	                  IF #coordSystem = #INDEX_COORDSYSTEM_TCS THEN
	                    #instMC_MoveLinearRelative.CoordSystem := "CS_WCS";
	                    IF #jogDirection < #JOG_DIRECTION_A THEN
	                      "LKinCtrl_OcsToWcs"(ocsX      := 0,
	                                          ocsY      := 0,
	                                          ocsZ      := 0,
	                                          ocsA      := #axesGroup.TcpInWcs.a.Position,
	                                          ocsB      := #axesGroup.TcpInWcs.b.Position,
	                                          ocsC      := #axesGroup.TcpInWcs.c.Position,
	                                          pointXOcs := #instMC_MoveLinearRelative.Distance[1],
	                                          pointYOcs := #instMC_MoveLinearRelative.Distance[2],
	                                          pointZOcs := #instMC_MoveLinearRelative.Distance[3],
	                                          pointAOcs := #instMC_MoveLinearRelative.Distance[4],
	                                          pointBOcs := #instMC_MoveLinearRelative.Distance[5],
	                                          pointCOcs := #instMC_MoveLinearRelative.Distance[6],
	                                          pointXWcs => #instMC_MoveLinearRelative.Distance[1],
	                                          pointYWcs => #instMC_MoveLinearRelative.Distance[2],
	                                          pointZWcs => #instMC_MoveLinearRelative.Distance[3],
	                                          pointAWcs => #instMC_MoveLinearRelative.Distance[4],
	                                          pointBWcs => #instMC_MoveLinearRelative.Distance[5],
	                                          pointCWcs => #instMC_MoveLinearRelative.Distance[6]);
	                      
	                      // reset rotation due to numeric inaccuracy of frame trans
	                      FOR #tempCounter := 4 TO 6 DO
	                        #instMC_MoveLinearRelative.Distance[#tempCounter] := 0.0;
	                      END_FOR;
	                    END_IF;
	                  ELSIF (#coordSystem >= "LKINCTRL_CS_NO_OF_FIRST_USER_FRAME" AND #coordSystem <= "LKINCTRL_CS_NO_OF_LAST_USER_FRAME") THEN
	                    #instMC_MoveLinearRelative.CoordSystem := "CS_WCS";
	                    IF #jogDirection < #JOG_DIRECTION_A THEN
	                      "LKinCtrl_OcsToWcs"(ocsX      := 0,
	                                          ocsY      := 0,
	                                          ocsZ      := 0,
	                                          ocsA      := #userFrames[#coordSystem].a,
	                                          ocsB      := #userFrames[#coordSystem].b,
	                                          ocsC      := #userFrames[#coordSystem].c,
	                                          pointXOcs := #instMC_MoveLinearRelative.Distance[1],
	                                          pointYOcs := #instMC_MoveLinearRelative.Distance[2],
	                                          pointZOcs := #instMC_MoveLinearRelative.Distance[3],
	                                          pointAOcs := #instMC_MoveLinearRelative.Distance[4],
	                                          pointBOcs := #instMC_MoveLinearRelative.Distance[5],
	                                          pointCOcs := #instMC_MoveLinearRelative.Distance[6],
	                                          pointXWcs => #instMC_MoveLinearRelative.Distance[1],
	                                          pointYWcs => #instMC_MoveLinearRelative.Distance[2],
	                                          pointZWcs => #instMC_MoveLinearRelative.Distance[3],
	                                          pointAWcs => #instMC_MoveLinearRelative.Distance[4],
	                                          pointBWcs => #instMC_MoveLinearRelative.Distance[5],
	                                          pointCWcs => #instMC_MoveLinearRelative.Distance[6]);
	                      
	                      // reset rotation due to numeric inaccuracy of frame trans
	                      FOR #tempCounter := 4 TO 6 DO
	                        #instMC_MoveLinearRelative.Distance[#tempCounter] := 0.0;
	                      END_FOR;
	                    END_IF;
	                  END_IF;
	                END_IF;
	                
	              #JOG_DIRECTION_RZ..#JOG_DIRECTION_RX: // Jogging around A,B,C
	                // set MC_MoveLinearAbsolute parameter
	                #instMC_MoveLinearAbsolute.Velocity := #dynamics.path.velocity;
	                #instMC_MoveLinearAbsolute.Acceleration := #dynamics.path.acceleration;
	                #instMC_MoveLinearAbsolute.Deceleration := #dynamics.path.deceleration;
	                #instMC_MoveLinearAbsolute.Jerk := #dynamics.path.jerk;
	                
	                // read current position and rotation matrix
	                CASE #coordSystem OF
	                  "CS_WCS", #INDEX_COORDSYSTEM_TCS: // in WCS and TCS
	                    // get rotation matrix representation of current position
	                    "LKinCtrl_RotXYZ"(angleA       := #axesGroup.TcpInWcs.a.Position,
	                                      angleB       := #axesGroup.TcpInWcs.b.Position,
	                                      angleC       := #axesGroup.TcpInWcs.c.Position,
	                                      resultMatrix := #statRotMatrix1);
	                    
	                    // do not move translatory
	                    #instMC_MoveLinearAbsolute.CoordSystem := "CS_WCS";
	                    #instMC_MoveLinearAbsolute.Position[1] := #axesGroup.TcpInWcs.x.Position;
	                    #instMC_MoveLinearAbsolute.Position[2] := #axesGroup.TcpInWcs.y.Position;
	                    #instMC_MoveLinearAbsolute.Position[3] := #axesGroup.TcpInWcs.z.Position;
	                  "CS_OCS1".."CS_OCS3": // OCS 1-3
	                    // get rotation matrix representation of current position
	                    "LKinCtrl_RotXYZ"(angleA       := #axesGroup.TcpInOcs[#coordSystem].a.Position,
	                                      angleB       := #axesGroup.TcpInOcs[#coordSystem].b.Position,
	                                      angleC       := #axesGroup.TcpInOcs[#coordSystem].c.Position,
	                                      resultMatrix := #statRotMatrix1);
	                    
	                    // do not move translatory
	                    #instMC_MoveLinearAbsolute.CoordSystem := #coordSystem;
	                    #instMC_MoveLinearAbsolute.Position[1] := #axesGroup.TcpInOcs[#coordSystem].x.Position;
	                    #instMC_MoveLinearAbsolute.Position[2] := #axesGroup.TcpInOcs[#coordSystem].y.Position;
	                    #instMC_MoveLinearAbsolute.Position[3] := #axesGroup.TcpInOcs[#coordSystem].z.Position;
	                  "LKINCTRL_CS_NO_OF_FIRST_USER_FRAME".."LKINCTRL_CS_NO_OF_LAST_USER_FRAME": // UCS
	                    // Calculate current UCS position 
	                    "LKinCtrl_WcsToOcs"(ocsX      := #userFrames[#coordSystem].x,
	                                        ocsY      := #userFrames[#coordSystem].y,
	                                        ocsZ      := #userFrames[#coordSystem].z,
	                                        ocsA      := #userFrames[#coordSystem].a,
	                                        ocsB      := #userFrames[#coordSystem].b,
	                                        ocsC      := #userFrames[#coordSystem].c,
	                                        pointXWcs := #axesGroup.TcpInWcs.x.Position,
	                                        pointYWcs := #axesGroup.TcpInWcs.y.Position,
	                                        pointZWcs := #axesGroup.TcpInWcs.z.Position,
	                                        pointAWcs := #axesGroup.TcpInWcs.a.Position,
	                                        pointBWcs := #axesGroup.TcpInWcs.b.Position,
	                                        pointCWcs := #axesGroup.TcpInWcs.c.Position,
	                                        pointXOcs => #tempTcpInUcs[1],
	                                        pointYOcs => #tempTcpInUcs[2],
	                                        pointZOcs => #tempTcpInUcs[3],
	                                        pointAOcs => #tempTcpInUcs[4],
	                                        pointBOcs => #tempTcpInUcs[5],
	                                        pointCOcs => #tempTcpInUcs[6]);
	                    
	                    // get rotation matrix representation of current position
	                    "LKinCtrl_RotXYZ"(angleA       := #tempTcpInUcs[4],
	                                      angleB       := #tempTcpInUcs[5],
	                                      angleC       := #tempTcpInUcs[6],
	                                      resultMatrix := #statRotMatrix1);
	                    
	                    // do not move translatory
	                    #instMC_MoveLinearAbsolute.CoordSystem := "CS_WCS";
	                    #instMC_MoveLinearAbsolute.Position[1] := #axesGroup.TcpInWcs.x.Position;
	                    #instMC_MoveLinearAbsolute.Position[2] := #axesGroup.TcpInWcs.y.Position;
	                    #instMC_MoveLinearAbsolute.Position[3] := #axesGroup.TcpInWcs.z.Position;
	                END_CASE;
	                
	                // Get rotation matrix based on direction and distance
	                CASE #jogDirection OF
	                  #JOG_DIRECTION_RZ:
	                    "LKinCtrl_RotZ"(angle     := #tempJogDistance,
	                                    rotMatrix := #statRotMatrix2);
	                  #JOG_DIRECTION_RY:
	                    "LKinCtrl_RotY"(angle     := #tempJogDistance,
	                                    rotMatrix := #statRotMatrix2);
	                  #JOG_DIRECTION_RX:
	                    "LKinCtrl_RotX"(angle     := #tempJogDistance,
	                                    rotMatrix := #statRotMatrix2);
	                END_CASE;
	                
	                // Calculate rotation matrix for target orientation
	                IF #coordSystem = #INDEX_COORDSYSTEM_TCS THEN
	                  // Calc rotation matrix TCS
	                  "LKinCtrl_MatrixMultiplication"(error        => #tempError,
	                                                  status       => #tempRetStatus,
	                                                  matrix1      := #statRotMatrix1,
	                                                  matrix2      := #statRotMatrix2,
	                                                  matrixResult := #statRotMatrix3);
	                ELSE
	                  // Calc rotation matrix regular
	                  "LKinCtrl_MatrixMultiplication"(error        => #tempError,
	                                                  status       => #tempRetStatus,
	                                                  matrix1      := #statRotMatrix2,
	                                                  matrix2      := #statRotMatrix1,
	                                                  matrixResult := #statRotMatrix3);
	                END_IF;
	                
	                // Assign target orientation to MC_MoveLinearAbsolute
	                IF #coordSystem >= "LKINCTRL_CS_NO_OF_FIRST_USER_FRAME" AND #coordSystem <= "LKINCTRL_CS_NO_OF_LAST_USER_FRAME" THEN
	                  // calculate rotated target position in UCS
	                  "LKinCtrl_InvRotXYZ"(A         => #tempTcpInUcs[4],
	                                       B         => #tempTcpInUcs[5],
	                                       C         => #tempTcpInUcs[6],
	                                       rotMatrix := #statRotMatrix3);
	                  
	                  // Calculate target WCS position since coordinate system of UCS for system is WCS
	                  "LKinCtrl_OcsToWcs"(ocsX      := #userFrames[#coordSystem].x,
	                                      ocsY      := #userFrames[#coordSystem].y,
	                                      ocsZ      := #userFrames[#coordSystem].z,
	                                      ocsA      := #userFrames[#coordSystem].a,
	                                      ocsB      := #userFrames[#coordSystem].b,
	                                      ocsC      := #userFrames[#coordSystem].c,
	                                      pointXOcs := #tempTcpInUcs[1],
	                                      pointYOcs := #tempTcpInUcs[2],
	                                      pointZOcs := #tempTcpInUcs[3],
	                                      pointAOcs := #tempTcpInUcs[4],
	                                      pointBOcs := #tempTcpInUcs[5],
	                                      pointCOcs := #tempTcpInUcs[6],
	                                      pointXWcs => #tempTcpInUcs[1], // dummy
	                                      pointYWcs => #tempTcpInUcs[2], // dummy
	                                      pointZWcs => #tempTcpInUcs[3], // dummy
	                                      pointAWcs => #instMC_MoveLinearAbsolute.Position[4],
	                                      pointBWcs => #instMC_MoveLinearAbsolute.Position[5],
	                                      pointCWcs => #instMC_MoveLinearAbsolute.Position[6]);
	                  
	                ELSE
	                  // calculate rotated target position
	                  "LKinCtrl_InvRotXYZ"(A         => #instMC_MoveLinearAbsolute.Position[4],
	                                       B         => #instMC_MoveLinearAbsolute.Position[5],
	                                       C         => #instMC_MoveLinearAbsolute.Position[6],
	                                       rotMatrix := #statRotMatrix3);
	                END_IF;
	                
	                // 3D + A,B plausibility check for C
	                IF #statTypeOfKinematics = 26 OR #statTypeOfKinematics = 27 OR #statTypeOfKinematics = 35 THEN
	                  // Check if C is around 0.0 or +-180.0
	                  IF ABS(180.0 - #instMC_MoveLinearAbsolute.Position[6]) < #TOLERANCE_C THEN // Check +180°
	                    #instMC_MoveLinearAbsolute.Position[6] := 180.0;
	                  ELSIF ABS(-180.0 - #instMC_MoveLinearAbsolute.Position[6]) < #TOLERANCE_C THEN // Check -180°
	                    #instMC_MoveLinearAbsolute.Position[6] := -180.0;
	                  ELSIF ABS(#instMC_MoveLinearAbsolute.Position[6]) < #TOLERANCE_C THEN // Check 0.0
	                    #instMC_MoveLinearAbsolute.Position[6] := 0.0;
	                  ELSE
	                    // error wrong value for C
	                    #statStatus := #ERR_JOG_DIRECTION_NOT_POSSIBLE;
	                  END_IF;
	                END_IF;
	                
	            END_CASE;
	            
	          END_REGION
	            // jog to position
	            //*********************************************************************************************************
	        ELSIF #tempJogToPosition THEN
	          REGION JOG_TO_TARGET_LINEAR
	            // set jog target position and configuration
	            #instMC_MoveLinearAbsolute.Position[1] := #targetPosition.x;
	            #instMC_MoveLinearAbsolute.Position[2] := #targetPosition.y;
	            #instMC_MoveLinearAbsolute.Position[3] := #targetPosition.z;
	            #instMC_MoveLinearAbsolute.Position[4] := #targetPosition.a;
	            #instMC_MoveLinearAbsolute.Position[5] := #targetPosition.b;
	            #instMC_MoveLinearAbsolute.Position[6] := #targetPosition.c;
	            #instMC_MoveLinearAbsolute.CoordSystem := #coordSystem;
	            // convert from UCS to WCS if necessary
	            IF (#coordSystem >= "LKINCTRL_CS_NO_OF_FIRST_USER_FRAME" AND #coordSystem <= "LKINCTRL_CS_NO_OF_LAST_USER_FRAME") THEN
	              #instMC_MoveLinearAbsolute.CoordSystem := "CS_WCS";
	              "LKinCtrl_OcsToWcs"(ocsX      := #userFrames[#coordSystem].x,
	                                  ocsY      := #userFrames[#coordSystem].y,
	                                  ocsZ      := #userFrames[#coordSystem].z,
	                                  ocsA      := #userFrames[#coordSystem].a,
	                                  ocsB      := #userFrames[#coordSystem].b,
	                                  ocsC      := #userFrames[#coordSystem].c,
	                                  pointXOcs := #targetPosition.x,
	                                  pointYOcs := #targetPosition.y,
	                                  pointZOcs := #targetPosition.z,
	                                  pointAOcs := #targetPosition.a,
	                                  pointBOcs := #targetPosition.b,
	                                  pointCOcs := #targetPosition.c,
	                                  pointXWcs => #instMC_MoveLinearAbsolute.Position[1],
	                                  pointYWcs => #instMC_MoveLinearAbsolute.Position[2],
	                                  pointZWcs => #instMC_MoveLinearAbsolute.Position[3],
	                                  pointAWcs => #instMC_MoveLinearAbsolute.Position[4],
	                                  pointBWcs => #instMC_MoveLinearAbsolute.Position[5],
	                                  pointCWcs => #instMC_MoveLinearAbsolute.Position[6]);
	            END_IF;
	            // convert from TCS to WCS if necessary
	            IF #coordSystem = #INDEX_COORDSYSTEM_TCS THEN
	              #instMC_MoveLinearAbsolute.CoordSystem := "CS_WCS";
	              "LKinCtrl_OcsToWcs"(ocsX      := #axesGroup.TcpInWcs.x.Position,
	                                  ocsY      := #axesGroup.TcpInWcs.y.Position,
	                                  ocsZ      := #axesGroup.TcpInWcs.z.Position,
	                                  ocsA      := #axesGroup.TcpInWcs.a.Position,
	                                  ocsB      := #axesGroup.TcpInWcs.b.Position,
	                                  ocsC      := #axesGroup.TcpInWcs.c.Position,
	                                  pointXOcs := #instMC_MoveLinearAbsolute.Position[1],
	                                  pointYOcs := #instMC_MoveLinearAbsolute.Position[2],
	                                  pointZOcs := #instMC_MoveLinearAbsolute.Position[3],
	                                  pointAOcs := #instMC_MoveLinearAbsolute.Position[4],
	                                  pointBOcs := #instMC_MoveLinearAbsolute.Position[5],
	                                  pointCOcs := #instMC_MoveLinearAbsolute.Position[6],
	                                  pointXWcs => #instMC_MoveLinearAbsolute.Position[1],
	                                  pointYWcs => #instMC_MoveLinearAbsolute.Position[2],
	                                  pointZWcs => #instMC_MoveLinearAbsolute.Position[3],
	                                  pointAWcs => #instMC_MoveLinearAbsolute.Position[4],
	                                  pointBWcs => #instMC_MoveLinearAbsolute.Position[5],
	                                  pointCWcs => #instMC_MoveLinearAbsolute.Position[6]);
	            END_IF;
	            
	            #instMC_MoveLinearAbsolute.Velocity := #dynamics.path.velocity;
	            #instMC_MoveLinearAbsolute.Acceleration := #dynamics.path.acceleration;
	            #instMC_MoveLinearAbsolute.Deceleration := #dynamics.path.deceleration;
	            #instMC_MoveLinearAbsolute.Jerk := #dynamics.path.jerk;
	            #instMC_MoveLinearAbsolute.DynamicAdaption := #dynamics.dynamicAdaption;
	            #instMC_MoveLinearAbsolute.DirectionA := #dynamics.directionA;
	          END_REGION
	            // jog synchronous point to point
	            //*********************************************************************************************************
	        ELSIF #tempJogSPTP THEN
	          REGION JOG_TO_POS_SPTP
	            #instMC_MoveDirectAbsolute.Position[1] := #targetPosition.x;
	            #instMC_MoveDirectAbsolute.Position[2] := #targetPosition.y;
	            #instMC_MoveDirectAbsolute.Position[3] := #targetPosition.z;
	            #instMC_MoveDirectAbsolute.Position[4] := #targetPosition.a;
	            #instMC_MoveDirectAbsolute.Position[5] := #targetPosition.b;
	            #instMC_MoveDirectAbsolute.Position[6] := #targetPosition.c;
	            #instMC_MoveDirectAbsolute.CoordSystem := #coordSystem;
	            // convert from UCS to WCS if necessary
	            IF (#coordSystem >= "LKINCTRL_CS_NO_OF_FIRST_USER_FRAME" AND #coordSystem <= "LKINCTRL_CS_NO_OF_LAST_USER_FRAME") THEN
	              #instMC_MoveDirectAbsolute.CoordSystem := "CS_WCS";
	              "LKinCtrl_OcsToWcs"(ocsX      := #userFrames[#coordSystem].x,
	                                  ocsY      := #userFrames[#coordSystem].y,
	                                  ocsZ      := #userFrames[#coordSystem].z,
	                                  ocsA      := #userFrames[#coordSystem].a,
	                                  ocsB      := #userFrames[#coordSystem].b,
	                                  ocsC      := #userFrames[#coordSystem].c,
	                                  pointXOcs := #targetPosition.x,
	                                  pointYOcs := #targetPosition.y,
	                                  pointZOcs := #targetPosition.z,
	                                  pointAOcs := #targetPosition.a,
	                                  pointBOcs := #targetPosition.b,
	                                  pointCOcs := #targetPosition.c,
	                                  pointXWcs => #instMC_MoveDirectAbsolute.Position[1],
	                                  pointYWcs => #instMC_MoveDirectAbsolute.Position[2],
	                                  pointZWcs => #instMC_MoveDirectAbsolute.Position[3],
	                                  pointAWcs => #instMC_MoveDirectAbsolute.Position[4],
	                                  pointBWcs => #instMC_MoveDirectAbsolute.Position[5],
	                                  pointCWcs => #instMC_MoveDirectAbsolute.Position[6]);
	            END_IF;
	            
	            #instMC_MoveDirectAbsolute.VelocityFactor := #dynamics.sPTP.velocityFactor;
	            #instMC_MoveDirectAbsolute.AccelerationFactor := #dynamics.sPTP.accelerationFactor;
	            #instMC_MoveDirectAbsolute.DecelerationFactor := #dynamics.sPTP.decelerationFactor;
	            #instMC_MoveDirectAbsolute.JerkFactor := #dynamics.sPTP.jerkFactor;
	            #instMC_MoveDirectAbsolute.LinkConstellation := #linkconstellation;
	            #instMC_MoveDirectAbsolute.PositionMode := 1;
	            #instMC_MoveDirectAbsolute.DirectionA := #dynamics.directionA;
	            #instMC_MoveDirectAbsolute.TurnJoint := #turnJoint;
	          END_REGION
	          END_IF;
	        END_REGION
	        
	        REGION SET_ORIENTATION_DYNAMICS
	          IF (((#jogDirection >= #JOG_DIRECTION_A AND #jogDirection <= #JOG_DIRECTION_RX) AND (#tempJogForward OR #tempJogBackward)) OR #tempJogToPosition)
	            AND (#dynamics.orientation.velocity > 0.0 // check if change of orientation dynamics is required
	            OR #dynamics.orientation.acceleration > 0.0
	            OR #dynamics.orientation.deceleration > 0.0
	            OR #dynamics.orientation.jerk > 0.0)
	          THEN
	            // safe default dynamics for orientation axis
	            #statOrientationDynamicsOld.velocity := #axesGroup.DynamicDefaults.Orientation.Velocity;
	            #statOrientationDynamicsOld.acceleration := #axesGroup.DynamicDefaults.Orientation.Acceleration;
	            #statOrientationDynamicsOld.deceleration := #axesGroup.DynamicDefaults.Orientation.Deceleration;
	            #statOrientationDynamicsOld.jerk := #axesGroup.DynamicDefaults.Orientation.Jerk;
	            
	            // change orientation default dynamics temporary
	            IF #dynamics.orientation.velocity > 0.0 THEN
	              #axesGroup.DynamicDefaults.Orientation.Velocity := #dynamics.orientation.velocity;
	            END_IF;
	            IF #dynamics.orientation.acceleration > 0.0 THEN
	              #axesGroup.DynamicDefaults.Orientation.Acceleration := #dynamics.orientation.acceleration;
	            END_IF;
	            IF #dynamics.orientation.deceleration > 0.0 THEN
	              #axesGroup.DynamicDefaults.Orientation.Deceleration := #dynamics.orientation.deceleration;
	            END_IF;
	            IF #dynamics.orientation.jerk > 0.0 THEN
	              #axesGroup.DynamicDefaults.Orientation.Jerk := #dynamics.orientation.jerk;
	            END_IF;
	            
	            // Orientation default dynamics will be reseted to previous values after jogging
	            #statOrientationDynamicsChanged := TRUE;
	          END_IF;
	        END_REGION
	        
	        REGION STATE_TRANSITION
	          IF (#statStatus <= #STATUS_SUBSEQUENT_CALL) THEN
	            // check if change of tool is required
	            IF (#tool <> #statToolOld) THEN
	              #statFBState := #FB_STATE_SET_TOOL;
	            ELSE // execute movement
	              #statFBState := #FB_STATE_EXECUTE_MOVEMENT;
	            END_IF;
	          ELSE
	            ;
	          END_IF;
	        END_REGION
	      END_IF;
	      
	    #FB_STATE_SET_TOOL:
	      REGION TOOL_CHANGE
	        IF #axesGroup.StatusWord.%X6 // no motion command is active
	          AND NOT #axesGroup.StatusWord.%X17 // not interrupted
	          AND #axesGroup.StatusWord.%X12 // constant velocity
	        THEN
	          #instMC_SetTool.Execute := TRUE;
	          #instMC_SetTool.ToolNumber := #tool;
	        END_IF;
	      END_REGION
	      
	      REGION STATE_TRANSITION
	        // tool has been changed
	        IF #instMC_SetTool.Done THEN
	          //#statToolOld := #tool;
	          #statFBState := #FB_STATE_EXECUTE_MOVEMENT;
	        END_IF;
	      END_REGION
	      
	    #FB_STATE_EXECUTE_MOVEMENT:
	      REGION SET_JOG_COMMAND
	        // Cartesian jogging
	        IF (#tempJogForward OR #tempJogBackward) THEN
	          IF #coordSystem = #INDEX_COORDSYSTEM_MCS OR #coordSystem = #INDEX_COORDSYSTEM_JCS THEN
	            #instMC_MoveDirectRelative.Execute := TRUE;
	          ELSE
	            IF #jogDirection < #JOG_DIRECTION_RZ THEN
	              #instMC_MoveLinearRelative.Execute := TRUE;
	            ELSE
	              #instMC_MoveLinearAbsolute.Execute := TRUE;
	            END_IF;
	          END_IF;
	          
	          // jog to target position  
	        ELSIF #tempJogToPosition THEN
	          #instMC_MoveLinearAbsolute.Execute := TRUE;
	          
	          //jog synchronous point to point
	        ELSIF #tempJogSPTP THEN
	          #instMC_MoveDirectAbsolute.Execute := TRUE;
	          
	        ELSE
	          #instMC_MoveLinearRelative.Execute := FALSE;
	          #instMC_MoveLinearAbsolute.Execute := FALSE;
	          #instMC_MoveDirectAbsolute.Execute := FALSE;
	          #instMC_MoveDirectRelative.Execute := FALSE;
	        END_IF;
	      END_REGION
	      
	      REGION STATE_TRANSITION
	        IF #instMC_MoveLinearRelative.Done
	          OR #instMC_MoveLinearAbsolute.Done
	          OR #instMC_MoveDirectAbsolute.Done
	          OR #instMC_MoveDirectRelative.Done
	        THEN
	          #statFBState := #FB_STATE_RESET_TOOL;
	          #statStatusBeforeResetTool := #STATUS_EXECUTION_FINISHED;
	        END_IF;
	      END_REGION
	      
	    #FB_STATE_STOP:
	      REGION STOP_KINEMATICS_MOTION
	        // set execute if group stop not busy
	        #instMC_GroupStop.Execute := (NOT #instMC_GroupStop.Busy AND NOT #instMC_GroupStop.Done AND NOT #instMC_GroupStop.Error AND #statStatus <> #STATUS_OUT_OF_JOINT_LIMITS);
	      END_REGION
	        
	      REGION STATE_TRANSITION
	        // save the errors or status until reset tool is done
	        IF (#instMC_GroupStop.Done AND #axesGroup.StatusWord.%X6) THEN // Added X6 according to AW
	          #statStatusBeforeResetTool := #STATUS_EXECUTION_FINISHED;
	        ELSIF #axesGroup.StatusWord.%X1 THEN // general TO error
	          #statStatusBeforeResetTool := #ERR_TO_KINEMATICS;
	          // Avoid error - 'job cannot be executed because a "MC_GroupStop" job is active' - 16#80CD - according to JH
	        ELSIF #instMC_MoveLinearRelative.Error AND #instMC_MoveLinearRelative.ErrorId <> 16#80CD THEN
	          #statStatusBeforeResetTool := #instMC_MoveLinearRelative.ErrorId;
	        ELSIF #instMC_MoveLinearAbsolute.Error AND #instMC_MoveLinearAbsolute.ErrorId <> 16#80CD THEN
	          #statStatusBeforeResetTool := #instMC_MoveLinearAbsolute.ErrorId;
	        ELSIF #instMC_MoveDirectAbsolute.Error AND #instMC_MoveDirectAbsolute.ErrorId <> 16#80CD THEN
	          #statStatusBeforeResetTool := #instMC_MoveDirectAbsolute.ErrorId;
	        ELSIF #instMC_MoveDirectRelative.Error AND #instMC_MoveDirectRelative.ErrorId <> 16#80CD THEN
	          #statStatusBeforeResetTool := #instMC_MoveDirectRelative.ErrorId;
	        ELSIF #instMC_SetTool.Error THEN
	          #statStatusBeforeResetTool := #instMC_SetTool.ErrorId;
	        ELSIF #instMC_GroupStop.Error THEN
	          #statStatusBeforeResetTool := #instMC_GroupStop.ErrorId;
	        ELSIF #statStatus = #STATUS_OUT_OF_JOINT_LIMITS THEN
	          #statStatusBeforeResetTool := #STATUS_EXECUTION_FINISHED;
	        END_IF;
	        
	        // reset tool as last step
	        IF (#instMC_GroupStop.Done AND #axesGroup.StatusWord.%X6)
	          OR #instMC_GroupStop.Error
	        THEN
	          #statFBState := #FB_STATE_RESET_TOOL;
	        END_IF;
	      END_REGION
	      
	    #FB_STATE_RESET_TOOL:
	      REGION RESET_TOOL
	        // any transition to FB_STATE_RESET_TOOL must set the statStatusBeforeResetTool
	        IF #tool <> #statToolOld THEN
	          IF #axesGroup.StatusWord.%X6 // no motion command is active
	            AND NOT #axesGroup.StatusWord.%X17 // not interrupted
	            AND #axesGroup.StatusWord.%X12 // constant velocity
	          THEN
	            #instMC_SetTool.Execute := TRUE;
	            #instMC_SetTool.ToolNumber := #statToolOld;
	          END_IF;
	          
	          IF #instMC_SetTool.Done OR #instMC_SetTool.Error THEN
	            #statStatus := #statStatusBeforeResetTool;
	          END_IF;
	        ELSE
	          #statStatus := #statStatusBeforeResetTool;
	        END_IF;
	      END_REGION
	      
	    ELSE // Undefined state in state machine reached
	      #statStatus := #ERR_UNDEFINED_STATE;
	  END_CASE;
	  
	END_REGION STATE_MACHINE
	
	REGION OUTPUTS
	  // Write outputs
	  IF (#statStatus = #STATUS_EXECUTION_FINISHED) AND (#statDone = FALSE) AND (#statError = FALSE) THEN // Execution finished without errors
	    #statDone := TRUE;
	    #statBusy := FALSE;
	    #statActive := FALSE;
	    #statError := FALSE;
	    #statFBState := #FB_STATE_NO_PROCESSING; // Switch state machine to "no processing"
	    
	  ELSIF (#statStatus.%X15 = TRUE) AND (#statError = FALSE) THEN // Error occurred (#statStatus is 16#8000 to 16#FFFF)
	    #statDone := FALSE;
	    #statBusy := FALSE;
	    #statActive := FALSE;
	    #statError := TRUE;
	    // Write diagnostics
	    #tempRet := RD_SYS_T(#diagnostics.timeStamp);
	    #diagnostics.stateNumber := #statFBState;
	    #diagnostics.status := #statStatus;
	    #statFBState := #FB_STATE_NO_PROCESSING; // Switch state machine to "no processing"
	    
	  ELSIF (#tempJogForward = FALSE AND #tempJogBackward = FALSE AND #tempJogToPosition = FALSE AND #tempJogSPTP = FALSE) AND ((#statDone = TRUE) OR (#statError = TRUE)) THEN // Reset outputs
	    #statDone := FALSE;
	    #statBusy := FALSE;
	    #statActive := FALSE;
	    #statError := FALSE;
	    #statStatus := #STATUS_NO_CALL;
	    #statJogForwardOld := FALSE;
	    #statJogBackwardOld := FALSE;
	    #statJogToPositionOld := FALSE;
	    #statJogSPTPOld := FALSE;
	  END_IF;
	  
	  // Write static values to outputs
	  #done := #statDone;
	  #busy := #statBusy;
	  #active := #statActive;
	  #error := #statError;
	  #status := #statStatus;
	  #remainingDistance := #statRemainingDistance;
	END_REGION OUTPUTS
	
	REGION CALL_FB_CYCLICALLY
	  // call FBs and set Execute = FALSE after the call
	  #instMC_GroupStop(AxesGroup := #axesGroup);
	  #instMC_GroupStop.Execute := FALSE;
	  
	  #instMC_MoveLinearAbsolute(AxesGroup := #axesGroup);
	  #instMC_MoveLinearAbsolute.Execute := FALSE;
	  
	  #instMC_MoveLinearRelative(AxesGroup := #axesGroup);
	  #instMC_MoveLinearRelative.Execute := FALSE;
	  
	  #instMC_SetTool(AxesGroup := #axesGroup);
	  #instMC_SetTool.Execute := FALSE;
	  
	  #instMC_MoveDirectAbsolute(AxesGroup := #axesGroup);
	  #instMC_MoveDirectAbsolute.Execute := FALSE;
	  
	  #instMC_MoveDirectRelative(AxesGroup := #axesGroup);
	  #instMC_MoveDirectRelative.Execute := FALSE;
	END_REGION
	
END_FUNCTION_BLOCK

FUNCTION "LKinCtrl_FramesValidValues" : Void
TITLE = LKinCtrl_FramesValidValues
{ S7_Optimized_Access := 'TRUE' }
AUTHOR : 'handling.team.automation@siemens.com'
FAMILY : LKinCtrl
VERSION : 5.0
   VAR_INPUT 
      mode : DInt;   // 0 = positioning, 1 = tool frame, 2 = OCS/KCS frame, 3 = MCS/JCS
      typeOfKinematics : DInt;   // Type of the TO_Kinematics (<TO>.Kinematics.TypeOfKinematics )
   END_VAR

   VAR_OUTPUT 
      frameCoordinateConfigurable : Array[0..5] of Bool;   // Determines if the offset/rotation by the coordinate is permitted
      upperLimitFrame : Array[0..5] of LReal;   // Upper limit of offset/rotation (exception: 3D with 2 orientation & mode positioning -> limits for C do not define a range but only these 2 values are allowed )
      lowerLimitFrame : Array[0..5] of LReal;   // Lower limit of the offset/rotation (exception: 3D with 2 orientation & mode positioning -> limits for C do not define a range but only these 2 values are allowed )
   END_VAR

   VAR_TEMP 
      tempCoordinatesCounter : DInt;   // Temporary variable to loop through the coordinates
      tempKinematicsType3D : DInt;   // Temporary variable to categorize the types of kinematics (2D, 2D with orientation, 3D, ...)
      tempFrameCoordinateConfigurable : Array[0..5] of Bool;   // Determines if the offset/rotation by the coordinate is permitted
      tempUpperLimitFrame : Array[0..5] of LReal;   // Upper limit of offset/rotation (exception: 3D with 2 orientation & mode positioning -> limits for C do not define a range but only these 2 values are allowed )
      tempLowerLimitFrame : Array[0..5] of LReal;   // Lower limit of the offset/rotation (exception: 3D with 2 orientation & mode positioning -> limits for C do not define a range but only these 2 values are allowed )
   END_VAR

   VAR CONSTANT 
      MODE_POSITIONING : DInt := 0;   // Mode returning the positioning frame limits
      MODE_TOOL_FRAME : DInt := 1;   // Mode returning the tool frame limits
      "MODE_OCS/KCS_FRAME" : DInt := 2;   // Mode returning the OCS/KCS frame limits
      "MODE_MCS/JCS_FRAME" : DInt := 3;   // Mode returning the MCS frame limits
      UPPER_LIMIT_MAX : LReal := 1000000000000.0;   // Maximum limit for the offset in x, y or z direction
      LOWER_LIMIT_MIN : LReal := -1000000000000.0;   // Minimum limit for the offset in x, y or z direction
   END_VAR


BEGIN
	//==========================================================================================
	// SIEMENS AG
	// (c)Copyright 2022 All Rights Reserved
	//------------------------------------------------------------------------------------------
	// Library: LKinCtrl
	// Tested with: S7-1517T-3 PN/DP
	// Engineering: TIA Portal V17
	// Restrictions: ---
	// Requirements: S7-1500T FW 2.9
	// Functionality: This FC returns the possible coordinates and ranges for a frame depending
	// on the kinematics type and the type of frame (positioning, tool frame, OCS/KCS frame).
	// Support: tech.team.motioncontrol@siemens.com
	// Note: Parameter comments are only available in language 'English (United States)'
	//------------------------------------------------------------------------------------------
	// Change log table:
	// Version    Date          Expert in charge    Changes applied
	// 01.00.00   14.12.2022    FF                  First created version
	// 01.00.01   09.02.2023    FF                  Added MCS/JCS (not limited), A is not limited
	//                                              for positioning of kinematics <= 4D
	//===========================================================================================
	
	//Categorize the different TO_Kinematics types
	CASE #typeOfKinematics OF
	  1, 5, 11, 15, 31:  // 2D kinematics
	    #tempKinematicsType3D := 1; // 1 - Cartesian portal 2D, Roller picker 2D, Articulated arm 2D, User-defined 2D
	  2, 6, 12, 16, 20, 32:  // 2D + orientation axis A
	    #tempKinematicsType3D := 2;   // 2 - Cartesian portal 2D with orientation, Roller picker 2D with orientation, Articulated arm 2D with orientation, Delta picker 2D with orientation, SCARA 2D with orientation, User-defined 2D with orientation A
	  3, 7, 13, 17, 21, 23, 33:  // 3D kinematics
	    #tempKinematicsType3D := 3;   // 3 - Cartesian portal 3D, Roller picker 3D (vertical), Articulated arm 3D, Delta picker 3D, Cylindrical robot 3D, Tripod 3D, User-defined 3D
	  4, 8, 9, 10, 14, 18, 22, 24, 34:  // 3D + orientation axis A
	    #tempKinematicsType3D := 4;   // 4 - Cartesian portal 3D with orientation, Roller picker 3D with orientation (vertical), Roller picker 3D with orientation (horizontal), SCARA 3D with orientation, Articulated arm 3D with orientation, Delta picker 3D with orientation, Cylindrical robot 3D with orientation, Tripod 3D with orientation, User-defined 3D with orientation A
	  26, 27, 35:// 3D + orientation axis A, B
	    #tempKinematicsType3D := 5;   // 5 - Cartesian portal 3D with 2 orientations A, B (Kin+), Delta picker 3D with 2 orientations A, B (Kin+), User-defined kinematics systems 3D with 2 orientations A, B (Kin+)
	  25, 36:// 3D + orientation axis A, B, C
	    #tempKinematicsType3D := 6;   // 6 - 6-axis articulated arm with central hand (Kin+), User-defined kinematics systems 3D with 3 orientations (Kin+)
	  ELSE  // invalid kinematics type
	    #tempKinematicsType3D := 0;
	END_CASE;
	//reset all outputs
	FOR #tempCoordinatesCounter := 0 TO 5 DO
	  #tempFrameCoordinateConfigurable[#tempCoordinatesCounter] := FALSE;
	  #tempUpperLimitFrame[#tempCoordinatesCounter] := 0.0;
	  #tempLowerLimitFrame[#tempCoordinatesCounter] := 0.0;
	END_FOR;
	//x coordinate
	IF (#mode = #MODE_TOOL_FRAME AND #tempKinematicsType3D <> 2) OR #mode <> #MODE_TOOL_FRAME THEN
	  #tempFrameCoordinateConfigurable[0] := TRUE;
	  #tempUpperLimitFrame[0] := #UPPER_LIMIT_MAX;
	  #tempLowerLimitFrame[0] := #LOWER_LIMIT_MIN;
	END_IF;
	//y coordinate
	IF #tempKinematicsType3D >= 3 OR #mode = #"MODE_MCS/JCS_FRAME" THEN
	  #tempFrameCoordinateConfigurable[1] := TRUE;
	  #tempUpperLimitFrame[1] := #UPPER_LIMIT_MAX;
	  #tempLowerLimitFrame[1] := #LOWER_LIMIT_MIN;
	END_IF;
	//z coordinate
	IF #mode <> #"MODE_MCS/JCS_FRAME" OR (#mode = #"MODE_MCS/JCS_FRAME" AND #tempKinematicsType3D >= 3) THEN
	  #tempFrameCoordinateConfigurable[2] := TRUE;
	  #tempUpperLimitFrame[2] := #UPPER_LIMIT_MAX;
	  #tempLowerLimitFrame[2] := #LOWER_LIMIT_MIN;
	END_IF;
	//a coordinate
	IF (#mode = #MODE_POSITIONING AND (#tempKinematicsType3D = 5 OR #tempKinematicsType3D = 6))
	  OR (#mode = #"MODE_OCS/KCS_FRAME" AND #tempKinematicsType3D >= 3)
	  OR (#mode = #MODE_TOOL_FRAME AND (#tempKinematicsType3D = 2 OR #tempKinematicsType3D = 4 OR #tempKinematicsType3D = 6)) THEN
	  #tempFrameCoordinateConfigurable[3] := TRUE;
	  #tempUpperLimitFrame[3] := 179.999;
	  #tempLowerLimitFrame[3] := -180.0;
	ELSIF (#mode = #MODE_POSITIONING AND (#tempKinematicsType3D = 2 OR #tempKinematicsType3D = 4))
	  OR (#mode = #"MODE_MCS/JCS_FRAME" AND (#tempKinematicsType3D = 2 OR #tempKinematicsType3D >= 4)) THEN
	  #tempFrameCoordinateConfigurable[3] := TRUE;
	  #tempUpperLimitFrame[3] := #UPPER_LIMIT_MAX;
	  #tempLowerLimitFrame[3] := #LOWER_LIMIT_MIN;
	END_IF;
	//b coordinate
	IF (#mode = #MODE_POSITIONING AND #tempKinematicsType3D >= 5)
	  OR (#mode = #MODE_TOOL_FRAME AND #tempKinematicsType3D = 6)
	  OR (#mode = #"MODE_OCS/KCS_FRAME" AND (#tempKinematicsType3D = 3 OR #tempKinematicsType3D = 6)) THEN
	  #tempFrameCoordinateConfigurable[4] := TRUE;
	  #tempUpperLimitFrame[4] := 90.0;
	  #tempLowerLimitFrame[4] := -90.0;
	ELSIF (#mode = #MODE_TOOL_FRAME AND #tempKinematicsType3D = 5)
	  OR (#mode = #"MODE_OCS/KCS_FRAME" AND #tempKinematicsType3D = 1) THEN
	  #tempFrameCoordinateConfigurable[4] := TRUE;
	  #tempUpperLimitFrame[4] := 179.999;
	  #tempLowerLimitFrame[4] := -180.0;
	ELSIF (#mode = #"MODE_MCS/JCS_FRAME" AND #tempKinematicsType3D >= 5) THEN
	  #tempFrameCoordinateConfigurable[4] := TRUE;
	  #tempUpperLimitFrame[4] := #UPPER_LIMIT_MAX;
	  #tempLowerLimitFrame[4] := #LOWER_LIMIT_MIN;
	END_IF;
	//c coordinate
	IF (#mode = #MODE_POSITIONING AND #tempKinematicsType3D = 6)
	  OR (#mode = #MODE_TOOL_FRAME AND #tempKinematicsType3D = 6)
	  OR (#mode = #"MODE_OCS/KCS_FRAME" AND (#tempKinematicsType3D = 3 OR #tempKinematicsType3D = 6)) THEN
	  #tempFrameCoordinateConfigurable[5] := TRUE;
	  #tempUpperLimitFrame[5] := 179.999;
	  #tempLowerLimitFrame[5] := -180.0;
	ELSIF #mode = #MODE_POSITIONING AND (#tempKinematicsType3D = 5) THEN // exception: limits do not define a range but only these 2 values are allowed
	  #tempFrameCoordinateConfigurable[5] := TRUE;
	  #tempUpperLimitFrame[5] := 0.0;
	  #tempLowerLimitFrame[5] := -180.0;
	ELSIF (#mode = #"MODE_MCS/JCS_FRAME" AND #tempKinematicsType3D = 6) THEN
	  #tempFrameCoordinateConfigurable[5] := TRUE;
	  #tempUpperLimitFrame[5] := #UPPER_LIMIT_MAX;
	  #tempLowerLimitFrame[5] := #LOWER_LIMIT_MIN;
	END_IF;
	//exceptions: SCARA 2D (OCS/KCS: offset in y direction and rotation around A are permissible)
	IF #mode = #"MODE_OCS/KCS_FRAME" AND #typeOfKinematics = 20 THEN
	  #tempFrameCoordinateConfigurable[1] := TRUE;
	  #tempUpperLimitFrame[1] := #UPPER_LIMIT_MAX;
	  #tempLowerLimitFrame[1] := #LOWER_LIMIT_MIN;
	  #tempFrameCoordinateConfigurable[3] := TRUE;
	  #tempUpperLimitFrame[3] := 179.999;
	  #tempLowerLimitFrame[3] := -180.0;
	END_IF;
	//outputs
	#frameCoordinateConfigurable := #tempFrameCoordinateConfigurable;
	#upperLimitFrame := #tempUpperLimitFrame;
	#lowerLimitFrame := #tempLowerLimitFrame;
END_FUNCTION

FUNCTION "LKinCtrl_OcsToWcs" : Void
TITLE = LKinCtrl_OcsToWcs
{ S7_Optimized_Access := 'TRUE' }
AUTHOR : 'handling.team.automation@siemens.com'
FAMILY : LKinCtrl
VERSION : 5.0
//Transfrom given position from OCS to WCS
   VAR_INPUT 
      ocsX : LReal;
      ocsY : LReal;
      ocsZ : LReal;
      ocsA : LReal;
      ocsB : LReal;
      ocsC : LReal;
      pointXOcs : LReal;
      pointYOcs : LReal;
      pointZOcs : LReal;
      pointAOcs : LReal;
      pointBOcs : LReal;
      pointCOcs : LReal;
   END_VAR

   VAR_OUTPUT 
      pointXWcs : LReal;
      pointYWcs : LReal;
      pointZWcs : LReal;
      pointAWcs : LReal;
      pointBWcs : LReal;
      pointCWcs : LReal;
   END_VAR

   VAR_TEMP 
      tempOcsTOcsP : Array[1..3, 1..1] of LReal;
      tempWcsTWcsOcs : Array[1..3, 1..1] of LReal;
      tempWcsTOcsP : Array[1..3, 1..1] of LReal;
      tempRWcsOcs : Array[1..3, 1..3] of LReal;
      tempROcsP : Array[1..3, 1..3] of LReal;
      tempRWcsP : Array[1..3, 1..3] of LReal;
      tempBool : Bool;
      tempWord : Word;
   END_VAR


BEGIN
	//=============================================================================
	// (company)
	// (c)Copyright (year)
	//-----------------------------------------------------------------------------
	// Library:       (that the source is dedicated to)
	// Tested with:   (test system with FW version)
	// Engineering:   TIA Portal (SW version)
	// Restrictions:  (OB types, etc.)
	// Requirements:  (hardware, technological package, memory needed, etc.)
	// Functionality: Transform a target position given in the OCS frame into an WCS frame
	//-----------------------------------------------------------------------------
	// Change log table:
	// Version  Date       Expert in charge Changes applied
	// 01.00.00 19.01.2022 JH               First released version
	//=============================================================================
	
	// input translation from OCS to P
	#tempOcsTOcsP[1, 1] := #pointXOcs;
	#tempOcsTOcsP[2, 1] := #pointYOcs;
	#tempOcsTOcsP[3, 1] := #pointZOcs;
	
	// input translation from WCS to OCS
	#tempWcsTWcsOcs[1, 1] := #ocsX;
	#tempWcsTWcsOcs[2, 1] := #ocsY;
	#tempWcsTWcsOcs[3, 1] := #ocsZ;
	
	// Create rotation matrix WCS in OCS
	// Rxyz(A,B,C) = [Rz(A) * Ry(B) * Rx(C)]
	"LKinCtrl_RotXYZ"(angleA := #ocsA,
	                  angleB := #ocsB,
	                  angleC := #ocsC,
	                  resultMatrix := #tempRWcsOcs);
	
	// Switch representation of point from OCS in WCS
	// Rxyz(A,B,C) * P
	"LKinCtrl_MatrixMultiplication"(status => #tempWord,
	                                matrix1 := #tempRWcsOcs,
	                                matrix2 := #tempOcsTOcsP,
	                                matrixResult := #tempWcsTOcsP,
	                                error => #tempBool);
	
	// Translational component
	#pointXWcs := #tempWcsTWcsOcs[1, 1] + #tempWcsTOcsP[1, 1];
	#pointYWcs := #tempWcsTWcsOcs[2, 1] + #tempWcsTOcsP[2, 1];
	#pointZWcs := #tempWcsTWcsOcs[3, 1] + #tempWcsTOcsP[3, 1];
	
	// Create rotation matrix OCS in Point
	// Rxyz(A,B,C) = Rz(A) * Ry(B) * Rx(C)
	"LKinCtrl_RotXYZ"(angleA := #pointAOcs,
	                  angleB := #pointBOcs,
	                  angleC := #pointCOcs,
	                  resultMatrix := #tempROcsP);
	
	// Rotation matrix WCS in Point
	"LKinCtrl_MatrixMultiplication"(status => #tempWord,
	                                matrix1 := #tempRWcsOcs,
	                                matrix2 := #tempROcsP,
	                                matrixResult := #tempRWcsP,
	                                error => #tempBool);
	
	// inverse problem from rotation matrix back to A,B,C
	"LKinCtrl_InvRotXYZ"(rotMatrix := #tempRWcsP,
	                     A => #pointAWcs,
	                     B => #pointBWcs,
	                     C => #pointCWcs);
	
	
END_FUNCTION

FUNCTION "LKinCtrl_RotXYZ" : Void
TITLE = LKinCtrl_RotXYZ
{ S7_Optimized_Access := 'TRUE' }
AUTHOR : 'handling.team.automation@siemens.com'
FAMILY : LKinCtrl
VERSION : 5.0
   VAR_INPUT 
      angleA : LReal;
      angleB : LReal;
      angleC : LReal;
   END_VAR

   VAR_IN_OUT 
      resultMatrix : Array[1..3, 1..3] of LReal;
   END_VAR

   VAR_TEMP 
      tempARad : LReal;
      tempBRad : LReal;
      tempCRad : LReal;
      tempDegRad : LReal;
   END_VAR

   VAR CONSTANT 
      PI : LReal := 3.14159265358979;
   END_VAR


BEGIN
	//=============================================================================
	// (company)
	// (c)Copyright (year)
	//-----------------------------------------------------------------------------
	// Library:       (that the source is dedicated to)
	// Tested with:   (test system with FW version)
	// Engineering:   TIA Portal (SW version)
	// Restrictions:  (OB types, etc.)
	// Requirements:  (hardware, technological package, memory needed, etc.)
	// Functionality: Calculate the rotation matrix for a fixed XYZ or current ZY'X'' rotation
	//-----------------------------------------------------------------------------
	// Change log table:
	// Version  Date       Expert in charge Changes applied
	// 01.00.00 19.01.2022 JH               First released version
	//=============================================================================
	#tempDegRad := #PI / 180.0;
	#tempARad := #angleA * #tempDegRad;
	#tempBRad := #angleB * #tempDegRad;
	#tempCRad := #angleC * #tempDegRad;
	
	// first column
	#resultMatrix[1, 1] := COS_LREAL(IN := #tempARad) * COS_LREAL(IN := #tempBRad);
	#resultMatrix[2, 1] := SIN_LREAL(IN := #tempARad) * COS_LREAL(IN := #tempBRad);
	#resultMatrix[3, 1] := - SIN_LREAL(IN := #tempBRad);
	
	// second column
	#resultMatrix[1, 2] := COS_LREAL(IN := #tempARad) * SIN_LREAL(IN := #tempBRad) * SIN_LREAL(IN := #tempCRad) - SIN_LREAL(IN := #tempARad) * COS_LREAL(IN := #tempCRad);
	#resultMatrix[2, 2] := SIN_LREAL(IN := #tempARad) * SIN_LREAL(IN := #tempBRad) * SIN_LREAL(IN := #tempCRad) + COS_LREAL(IN := #tempARad) * COS_LREAL(IN := #tempCRad);
	#resultMatrix[3, 2] := COS_LREAL(IN := #tempBRad) * SIN_LREAL(IN := #tempCRad);
	
	// third column
	#resultMatrix[1, 3] := COS_LREAL(IN := #tempARad) * SIN_LREAL(IN := #tempBRad) * COS_LREAL(IN := #tempCRad) + SIN_LREAL(IN := #tempARad) * SIN_LREAL(IN := #tempCRad);
	#resultMatrix[2, 3] := SIN_LREAL(IN := #tempARad) * SIN_LREAL(IN := #tempBRad) * COS_LREAL(IN := #tempCRad) - COS_LREAL(IN := #tempARad) * SIN_LREAL(IN := #tempCRad);
	#resultMatrix[3, 3] := COS_LREAL(IN := #tempBRad) * COS_LREAL(IN := #tempCRad);
END_FUNCTION

FUNCTION "LKinCtrl_MatrixMultiplication" : Void
TITLE = LKinCtrl_MatrixMultiplication
{ S7_Optimized_Access := 'TRUE' }
AUTHOR : 'handling.team.automation@siemens.com'
FAMILY : LKinCtrl
VERSION : 5.0
//Multiply given matrix 1 and 2 
   VAR_OUTPUT 
      error : Bool;
      status : Word;
   END_VAR

   VAR_IN_OUT 
      matrix1 : Array[*, *] of LReal;
      matrix2 : Array[*, *] of LReal;
      matrixResult : Array[*, *] of LReal;
   END_VAR

   VAR_TEMP 
      tempMatrix1LowerBoundRows : DInt;
      tempMatrix1LowerBoundColumns : DInt;
      tempMatrix1UpperBoundRows : DInt;
      tempMatrix1UpperBoundColumns : DInt;
      tempMatrix2LowerBoundRows : DInt;
      tempMatrix2LowerBoundColumns : DInt;
      tempMatrix2UpperBoundRows : DInt;
      tempMatrix2UpperBoundColumns : DInt;
      tempResultMatrixLowerBoundRows : DInt;
      tempResultMatrixLowerBoundColumns : DInt;
      tempResultMatrixUpperBoundRows : DInt;
      tempResultMatrixUpperBoundColumns : DInt;
      tempJ : DInt;
      tempK : DInt;
      tempL : DInt;
      tempResult : LReal;
   END_VAR

   VAR CONSTANT 
      ZERO : Real := 0.0;
      ROWS : UInt := 1;
      COLUMNS : UInt := 2;
      STATUS_NO_ERROR : Word := 16#0000;
      ERR_MATR1_LOWBOUND_COLUMNS_MATR2_LOWBOUND_ROWS : Word := 16#8200;
      ERR_MATR1_UPPBOUND_COLUMNS_MATR2_UPPBOUND_ROWS : Word := 16#8201;
      ERR_MATR1_LOWBOUND_ROWS_RESMATR_LOWBOUND_ROWS : Word := 16#8202;
      ERR_MATR2_LOWBOUND_COLUMNS_RESMATR_LOWBOUND_COLUMNS : Word := 16#8203;
      ERR_MATR1_UPPBOUND_ROWS_RESMATR_UPPBOUND_ROWS : Word := 16#8204;
      ERR_MATR2_UPPBOUND_COLUMNS_RESMATR_UPPBOUND_COLUMNS : Word := 16#8205;
   END_VAR


BEGIN
	REGION Block info header
	  //=============================================================================
	  // SIEMENS AG / (c)Copyright 2017
	  //-------------------------------------------------------------------------------
	  // Title:            LGF_MatrixMultiplication
	  // Comment/Function: Caluclates the multiplication of two matrices
	  // Library/Family:   LGF(Library General Functions)
	  // Author:           Siemens Digital Industry Support
	  // Tested with:      S7-PLCSIM Advanced V2.0 SP1
	  // Engineering:      TIA Portal V15 Update 2
	  // Restrictions:     ENO disabled - error handling done by error and status
	  // Requirements:     PLC (S7-1200 / S7-1500)
	  //-------------------------------------------------------------------------------
	  // Change log table:
	  // Version  | Date       | Expert in charge       | Changes applied
	  //----------|------------|------------------------|------------------------------
	  // 01.00.00 19.08.2015  Siemens Industry Online Support
	  //                      First released version
	  // 01.00.01 02.01.2017  Siemens Industry Online Support
	  //                      Upgrade: TIA Portal V14 Update 1
	  // 02.00.00 06.02.2017  Siemens Industry Online Support
	  //                      Functionality using Array[*,*]
	  // 02.00.01 17.08.2018  Siemens Industry Online Support
	  //                      Upgrade: TIA V15 Update 2
	  // 02.00.02 23.11.2018  Siemens Industry Online Support
	  //                      Upgrade: TIA V15.1
	  // 02.00.06 13.11.2019  Simatic Systems Support
	  //                      Regions, comments and constants are added
	  //                      Moved matrices to IO field.
	  // 03.00.00 23.04.2020  Simatic Systems Support
	  //                      Set version to V3.0.0, harmonize the version of the whole library
	  // 03.00.01 02.02.2020  Simatic Systems Support
	  //                      Insert documentation
	  //=================================================================================
	END_REGION Block info header
	
	REGION Getting matrices size
	  //Determine the size of the matrices
	  // Lower bound rows
	  #tempMatrix1LowerBoundRows := LOWER_BOUND(ARR := #matrix1, DIM := #ROWS);
	  #tempMatrix2LowerBoundRows := LOWER_BOUND(ARR := #matrix2, DIM := #ROWS);
	  #tempResultMatrixLowerBoundRows := LOWER_BOUND(ARR := #matrixResult, DIM := #ROWS);
	  // Lower bound columns
	  #tempMatrix1LowerBoundColumns := LOWER_BOUND(ARR := #matrix1, DIM := #COLUMNS);
	  #tempMatrix2LowerBoundColumns := LOWER_BOUND(ARR := #matrix2, DIM := #COLUMNS);
	  #tempResultMatrixLowerBoundColumns := LOWER_BOUND(ARR := #matrixResult, DIM := #COLUMNS);
	  
	  // Upper bound rows
	  #tempMatrix1UpperBoundRows := UPPER_BOUND(ARR := #matrix1, DIM := #ROWS);
	  #tempMatrix2UpperBoundRows := UPPER_BOUND(ARR := #matrix2, DIM := #ROWS);
	  #tempResultMatrixUpperBoundRows := UPPER_BOUND(ARR := #matrixResult, DIM := #ROWS);
	  // Upper bound columns
	  #tempMatrix1UpperBoundColumns := UPPER_BOUND(ARR := #matrix1, DIM := #COLUMNS);
	  #tempMatrix2UpperBoundColumns := UPPER_BOUND(ARR := #matrix2, DIM := #COLUMNS);
	  #tempResultMatrixUpperBoundColumns := UPPER_BOUND(ARR := #matrixResult, DIM := #COLUMNS);
	END_REGION
	
	REGION Error evaluation of matrices dimentions
	  // Matrix one must have the same count of rows as matrix two has columns. Else the multiplication is not possible.
	  IF #tempMatrix1LowerBoundColumns <> #tempMatrix2LowerBoundRows THEN
	    #error := true;
	    #status := #ERR_MATR1_LOWBOUND_COLUMNS_MATR2_LOWBOUND_ROWS;
	    RETURN;
	  ELSIF #tempMatrix1UpperBoundColumns <> #tempMatrix2UpperBoundRows THEN
	    #error := true;
	    #status := #ERR_MATR1_UPPBOUND_COLUMNS_MATR2_UPPBOUND_ROWS;
	    RETURN;
	  END_IF;
	  // Result matrix must have the same number of rows as matrix 1 and the same number of columns as the matrix 2.
	  IF (#tempMatrix1LowerBoundRows <> #tempResultMatrixLowerBoundRows) THEN
	    #error := true;
	    #status := #ERR_MATR1_LOWBOUND_ROWS_RESMATR_LOWBOUND_ROWS;
	    RETURN;
	  ELSIF (#tempMatrix1UpperBoundRows <> #tempResultMatrixUpperBoundRows) THEN
	    #error := true;
	    #status := #ERR_MATR1_UPPBOUND_ROWS_RESMATR_UPPBOUND_ROWS;
	    RETURN;
	  ELSIF (#tempMatrix2LowerBoundColumns <> #tempResultMatrixLowerBoundColumns) THEN
	    #error := true;
	    #status := #ERR_MATR2_LOWBOUND_COLUMNS_RESMATR_LOWBOUND_COLUMNS;
	    RETURN;
	  ELSIF (#tempMatrix2UpperBoundColumns <> #tempResultMatrixUpperBoundColumns) THEN
	    #error := true;
	    #status := #ERR_MATR2_UPPBOUND_COLUMNS_RESMATR_UPPBOUND_COLUMNS;
	    RETURN;
	  END_IF;
	END_REGION
	
	REGION Multiplication
	  //Multiplies each row with each column
	  FOR #tempJ := #tempMatrix1LowerBoundRows TO #tempMatrix1UpperBoundRows DO
	    FOR #tempK := #tempMatrix2LowerBoundColumns TO #tempMatrix2UpperBoundColumns DO
	      #tempResult := #ZERO;
	      FOR #tempL := #tempMatrix1LowerBoundColumns TO #tempMatrix1UpperBoundColumns DO
	        #tempResult := #tempResult + #matrix1[#tempJ, #tempL] * #matrix2[#tempL, #tempK];
	      END_FOR;
	      #matrixResult[#tempJ, #tempK] := #tempResult;
	    END_FOR;
	  END_FOR;
	  
	  #error := false;
	  #status := #STATUS_NO_ERROR;
	  // ENO mechanism is not used
	  ENO := TRUE;
	END_REGION
	
END_FUNCTION

FUNCTION "LKinCtrl_InvRotXYZ" : Void
TITLE = LKinCtrl_InvRotXYZ
{ S7_Optimized_Access := 'TRUE' }
AUTHOR : 'handling.team.automation@siemens.com'
FAMILY : LKinCtrl
VERSION : 5.0
//Given a rotation matrix, calculate the Euler angles A, B and C for an XYZ (ZY'X'') rotation
   VAR_OUTPUT 
      A : LReal;
      B : LReal;
      C : LReal;
   END_VAR

   VAR_IN_OUT 
      rotMatrix : Array[1..3, 1..3] of LReal;
   END_VAR

   VAR_TEMP 
      tempARadians : LReal;
      tempBRadians : LReal;
      tempCRadians : LReal;
      tempStatus : Word;
      tempError : Bool;
      tempRadDeg : LReal;
   END_VAR

   VAR CONSTANT 
      PI : LReal := 3.14159265358979;
   END_VAR


BEGIN
	//=============================================================================
	// (company)
	// (c)Copyright (year)
	//-----------------------------------------------------------------------------
	// Library:       (that the source is dedicated to)
	// Tested with:   (test system with FW version)
	// Engineering:   TIA Portal (SW version)
	// Restrictions:  (OB types, etc.)
	// Requirements:  (hardware, technological package, memory needed, etc.)
	// Functionality: Given a rotation matrix, calculate the Euler angles A, B and C for an XYZ (ZY'X'') rotation
	//-----------------------------------------------------------------------------
	// Change log table:
	// Version  Date       Expert in charge Changes applied
	// 01.00.00 19.01.2022 JH               First released version
	//=============================================================================
	
	IF NOT (#rotMatrix[3, 1] = 1) AND NOT (#rotMatrix[3, 1] = -1) THEN // no gimbal lock
	  
	  #tempBRadians := "LKinCtrl_ATan2"(opp := - #rotMatrix[3, 1],
	                                    adj := SQRT_LREAL(IN := (SQR_LREAL(IN := #rotMatrix[3, 2]) + SQR_LREAL(IN := #rotMatrix[3, 3]))));
	  
	  #tempARadians := "LKinCtrl_ATan2"(opp := #rotMatrix[2, 1],
	                                    adj := #rotMatrix[1, 1]);
	  
	  #tempCRadians := "LKinCtrl_ATan2"(opp := #rotMatrix[3, 2],
	                                    adj := #rotMatrix[3, 3]);
	ELSE // gimbal lock
	  #tempCRadians := 0; // arbitrarily choosen
	  IF #rotMatrix[3, 1] = -1 THEN // B = 90°
	    #tempBRadians := #PI / 2.0;
	    #tempARadians := - "LKinCtrl_ATan2"(opp := #rotMatrix[1, 2], adj := #rotMatrix[2, 2]);
	  ELSE // B = -90°
	    #tempBRadians := - #PI / 2.0;
	    #tempARadians := - "LKinCtrl_ATan2"(opp := #rotMatrix[1, 2], adj := #rotMatrix[2, 2]);
	  END_IF;
	END_IF;
	
	#tempRadDeg := 180.0 / #PI;
	#A := #tempARadians * #tempRadDeg;
	#B := #tempBRadians * #tempRadDeg;
	#C := #tempCRadians * #tempRadDeg;
	
	IF #A = 180.0 THEN
	  #A := - 180.0;
	END_IF;
	
	IF #C = 180.0 THEN
	  #C := - 180.0;
	END_IF;
	
END_FUNCTION

FUNCTION "LKinCtrl_ATan2" : LReal
TITLE = LKinCtrl_ATan2
{ S7_Optimized_Access := 'TRUE' }
AUTHOR : 'handling.team.automation@siemens.com'
FAMILY : LKinCtrl
VERSION : 5.0
   VAR_INPUT 
      opp : LReal;
      adj : LReal;
   END_VAR

   VAR CONSTANT 
      PI : LReal := 3.14159265358979;
      TOL_POS : LReal := 1.0E-09;
      TOL_NEG : LReal := -1.0E-09;
   END_VAR


BEGIN
	//=============================================================================
	// SIEMENS AG
	// (c)Copyright 2018 All Rights Reserved
	//-----------------------------------------------------------------------------
	// Library: LKinTrans 
	// Tested with: S7-1516T-3 PN
	// Engineering: TIA Portal V15
	// Restrictions: -
	// Requirements: S7-1500/S7-1500T FW 2.5
	// Functionality: Calculate arcTan2 (tan with definition -pi...pi)
	// Support: tech.team.motioncontrol@siemens.com
	// Note: Parameter comments are only available in language 'English (United States)'
	//-----------------------------------------------------------------------------
	// Change log table:
	// Version  Date       Expert in charge Changes applied
	// 01.00.00 02.07.2018 SF               created
	//=============================================================================
	
	// Calc values
	IF (#adj >= #TOL_POS) THEN
	  //first or forth quadrant
	  #LKinCtrl_ATan2 := ATAN(#opp / #adj);
	ELSIF (ABS(#adj) < #TOL_POS) THEN
	  IF (#opp >= #TOL_POS) THEN
	    //between first and second
	    #LKinCtrl_ATan2 := 0.5 * #PI;
	  ELSIF (#opp <= #TOL_NEG) THEN
	    //between third and forth
	    #LKinCtrl_ATan2 := -0.5 * #PI;
	  ELSE
	    //error - both components zero
	    #LKinCtrl_ATan2 := 0.0;
	  END_IF;
	ELSE //(#adj < 0.0) 
	  IF (#opp >= #TOL_POS) THEN
	    //second quadrant
	    #LKinCtrl_ATan2 := #PI + ATAN(#opp / #adj);
	  ELSIF (#opp <= #TOL_NEG) THEN
	    //third quadrant
	    #LKinCtrl_ATan2 := - #PI + ATAN(#opp / #adj);
	  ELSE
	    #LKinCtrl_ATan2 := - #PI;
	  END_IF;
	END_IF;
	
	
END_FUNCTION

FUNCTION "LKinCtrl_WcsToOcs" : Void
TITLE = LKinCtrl_WcsToOcs
{ S7_Optimized_Access := 'TRUE' }
AUTHOR : 'handling.team.automation@siemens.com'
FAMILY : LKinCtrl
VERSION : 5.0
   VAR_INPUT 
      ocsX : LReal;
      ocsY : LReal;
      ocsZ : LReal;
      ocsA : LReal;
      ocsB : LReal;
      ocsC : LReal;
      pointXWcs : LReal;
      pointYWcs : LReal;
      pointZWcs : LReal;
      pointAWcs : LReal;
      pointBWcs : LReal;
      pointCWcs : LReal;
   END_VAR

   VAR_OUTPUT 
      pointXOcs : LReal;
      pointYOcs : LReal;
      pointZOcs : LReal;
      pointAOcs : LReal;
      pointBOcs : LReal;
      pointCOcs : LReal;
   END_VAR

   VAR_TEMP 
      tempWcsTOcsP : Array[1..3, 1..1] of LReal;
      tempOcsTOcsP : Array[1..3, 1..1] of LReal;
      tempROcsWcs : Array[1..3, 1..3] of LReal;
      tempRWcsP : Array[1..3, 1..3] of LReal;
      tempROcsP : Array[1..3, 1..3] of LReal;
      tempBool : Bool;
      tempWord : Word;
   END_VAR


BEGIN
	//=============================================================================
	// (company)
	// (c)Copyright (year)
	//-----------------------------------------------------------------------------
	// Library:       (that the source is dedicated to)
	// Tested with:   (test system with FW version)
	// Engineering:   TIA Portal (SW version)
	// Restrictions:  (OB types, etc.)
	// Requirements:  (hardware, technological package, memory needed, etc.)
	// Functionality: Transform a target position given in the WCS frame into an OCS frame
	//-----------------------------------------------------------------------------
	// Change log table:
	// Version  Date       Expert in charge Changes applied
	// 01.00.00 19.01.2022 JH               First released version
	//=============================================================================
	
	// input translation from WCS to P
	#tempWcsTOcsP[1, 1] := #pointXWcs - #ocsX;
	#tempWcsTOcsP[2, 1] := #pointYWcs - #ocsY;
	#tempWcsTOcsP[3, 1] := #pointZWcs - #ocsZ;
	
	// Create rotation matrix OCS in WCS
	// Rxyz(A,B,C) = [Rz(A) * Ry(B) * Rx(C)]^T
	"LKinCtrl_RotXYZTranspose"(angleA := #ocsA,
	                           angleB := #ocsB,
	                           angleC := #ocsC,
	                           resultMatrix := #tempROcsWcs);
	
	// Switch representation of point from WCS in OCS
	// Rxyz(A,B,C) * P
	"LKinCtrl_MatrixMultiplication"(status => #tempWord,
	                                matrix1 := #tempROcsWcs,
	                                matrix2 := #tempWcsTOcsP,
	                                matrixResult := #tempOcsTOcsP,
	                                error => #tempBool);
	
	// Translational component
	#pointXOcs := #tempOcsTOcsP[1, 1];
	#pointYOcs := #tempOcsTOcsP[2, 1];
	#pointZOcs := #tempOcsTOcsP[3, 1];
	
	// Create rotation matrix WCS in Point
	// Rxyz(A,B,C) = Rz(A) * Ry(B) * Rx(C)
	"LKinCtrl_RotXYZ"(angleA := #pointAWcs,
	                  angleB := #pointBWcs,
	                  angleC := #pointCWcs,
	                  resultMatrix := #tempRWcsP);
	
	// Rotation matrix OCS in Point
	"LKinCtrl_MatrixMultiplication"(status => #tempWord,
	                                matrix1 := #tempROcsWcs,
	                                matrix2 := #tempRWcsP,
	                                matrixResult := #tempROcsP,
	                                error => #tempBool);
	
	// inverse problem from rotation matrix back to A,B,C
	"LKinCtrl_InvRotXYZ"(rotMatrix := #tempROcsP,
	                     A => #pointAOcs,
	                     B => #pointBOcs,
	                     C => #pointCOcs);
	
	
END_FUNCTION

FUNCTION "LKinCtrl_RotXYZTranspose" : Void
TITLE = LKinCtrl_RotXYZTranspose
{ S7_Optimized_Access := 'TRUE' }
AUTHOR : 'handling.team.automation@siemens.com'
FAMILY : LKinCtrl
VERSION : 5.0
   VAR_INPUT 
      angleA : LReal;
      angleB : LReal;
      angleC : LReal;
   END_VAR

   VAR_IN_OUT 
      resultMatrix : Array[1..3, 1..3] of LReal;
   END_VAR

   VAR_TEMP 
      tempARad : LReal;
      tempBRad : LReal;
      tempCRad : LReal;
      tempDegRad : LReal;
   END_VAR

   VAR CONSTANT 
      PI : LReal := 3.14159265358979;
   END_VAR


BEGIN
	//=============================================================================
	// (company)
	// (c)Copyright (year)
	//-----------------------------------------------------------------------------
	// Library:       (that the source is dedicated to)
	// Tested with:   (test system with FW version)
	// Engineering:   TIA Portal (SW version)
	// Restrictions:  (OB types, etc.)
	// Requirements:  (hardware, technological package, memory needed, etc.)
	// Functionality: Calculate the transpose rotation matrix for a fixed XYZ or current ZY'X'' rotation
	//-----------------------------------------------------------------------------
	// Change log table:
	// Version  Date       Expert in charge Changes applied
	// 01.00.00 19.01.2022 JH               First released version
	//=============================================================================
	
	#tempDegRad := #PI / 180.0;
	#tempARad := #angleA * #tempDegRad;
	#tempBRad := #angleB * #tempDegRad;
	#tempCRad := #angleC * #tempDegRad;
	
	
	// first row
	#resultMatrix[1, 1] := COS_LREAL(IN := #tempARad) * COS_LREAL(IN := #tempBRad);
	#resultMatrix[1, 2] := SIN_LREAL(IN := #tempARad) * COS_LREAL(IN := #tempBRad);
	#resultMatrix[1, 3] := - SIN_LREAL(IN := #tempBRad);
	
	// second row
	#resultMatrix[2, 1] := COS_LREAL(IN := #tempARad) * SIN_LREAL(IN := #tempBRad) * SIN_LREAL(IN := #tempCRad) - SIN_LREAL(IN := #tempARad) * COS_LREAL(IN := #tempCRad);
	#resultMatrix[2, 2] := SIN_LREAL(IN := #tempARad) * SIN_LREAL(IN := #tempBRad) * SIN_LREAL(IN := #tempCRad) + COS_LREAL(IN := #tempARad) * COS_LREAL(IN := #tempCRad);
	#resultMatrix[2, 3] := COS_LREAL(IN := #tempBRad) * SIN_LREAL(IN := #tempCRad);
	
	// third row
	#resultMatrix[3, 1] := COS_LREAL(IN := #tempARad) * SIN_LREAL(IN := #tempBRad) * COS_LREAL(IN := #tempCRad) + SIN_LREAL(IN := #tempARad) * SIN_LREAL(IN := #tempCRad);
	#resultMatrix[3, 2] := SIN_LREAL(IN := #tempARad) * SIN_LREAL(IN := #tempBRad) * COS_LREAL(IN := #tempCRad) - COS_LREAL(IN := #tempARad) * SIN_LREAL(IN := #tempCRad);
	#resultMatrix[3, 3] := COS_LREAL(IN := #tempBRad) * COS_LREAL(IN := #tempCRad);
END_FUNCTION

FUNCTION "LKinCtrl_RotZ" : Void
TITLE = LKinCtrl_RotZ
{ S7_Optimized_Access := 'TRUE' }
AUTHOR : 'handling.team.automation@siemens.com'
FAMILY : LKinCtrl
VERSION : 5.0
   VAR_INPUT 
      angle : LReal;
   END_VAR

   VAR_IN_OUT 
      rotMatrix : Array[1..3, 1..3] of LReal;
   END_VAR

   VAR_TEMP 
      tempAngleRadians : LReal;
   END_VAR

   VAR CONSTANT 
      PI : LReal := 3.14159265358979;   // Pi
   END_VAR


BEGIN
	// Rotationsmatrizen
	// RotZ:
	#tempAngleRadians := #angle * #PI / 180.0;
	
	// First row
	#rotMatrix[1, 1] := COS_LREAL(IN := #tempAngleRadians);
	#rotMatrix[1, 2] := - SIN_LREAL(IN := #tempAngleRadians);
	#rotMatrix[1, 3] := 0;
	
	// Second row
	#rotMatrix[2, 1] := SIN_LREAL(IN := #tempAngleRadians);
	#rotMatrix[2, 2] := COS_LREAL(IN := #tempAngleRadians);
	#rotMatrix[2, 3] := 0;
	
	// Third row
	#rotMatrix[3, 1] := 0;
	#rotMatrix[3, 2] := 0;
	#rotMatrix[3, 3] := 1;
END_FUNCTION

FUNCTION "LKinCtrl_RotY" : Void
TITLE = LKinCtrl_RotY
{ S7_Optimized_Access := 'TRUE' }
AUTHOR : 'handling.team.automation@siemens.com'
FAMILY : LKinCtrl
VERSION : 5.0
   VAR_INPUT 
      angle : LReal;
   END_VAR

   VAR_IN_OUT 
      rotMatrix : Array[1..3, 1..3] of LReal;
   END_VAR

   VAR_TEMP 
      tempAngleRadians : LReal;
   END_VAR

   VAR CONSTANT 
      PI : LReal := 3.14159265358979;   // Pi
   END_VAR


BEGIN
	// Rotationsmatrizen
	// RotY:
	#tempAngleRadians := #angle * #PI / 180.0;
	
	// First row
	#rotMatrix[1, 1] := COS_LREAL(IN := #tempAngleRadians);
	#rotMatrix[1, 2] := 0;
	#rotMatrix[1, 3] := SIN_LREAL(IN := #tempAngleRadians);
	
	// Second row
	#rotMatrix[2, 1] := 0;
	#rotMatrix[2, 2] := 1;
	#rotMatrix[2, 3] := 0;
	
	// Third row
	#rotMatrix[3, 1] := - SIN_LREAL(IN := #tempAngleRadians);
	#rotMatrix[3, 2] := 0;
	#rotMatrix[3, 3] := COS_LREAL(IN := #tempAngleRadians);
END_FUNCTION

FUNCTION "LKinCtrl_RotX" : Void
TITLE = LKinCtrl_RotX
{ S7_Optimized_Access := 'TRUE' }
AUTHOR : 'handling.team.automation@siemens.com'
FAMILY : LKinCtrl
VERSION : 5.0
   VAR_INPUT 
      angle : LReal;
   END_VAR

   VAR_IN_OUT 
      rotMatrix : Array[1..3, 1..3] of LReal;
   END_VAR

   VAR_TEMP 
      tempAngleRadians : LReal;
   END_VAR

   VAR CONSTANT 
      PI : LReal := 3.14159265358979;   // Pi
   END_VAR


BEGIN
	// Rotationsmatrizen
	// RotX:
	#tempAngleRadians := #angle * #PI / 180.0;
	
	// First row
	#rotMatrix[1, 1] := 1;
	#rotMatrix[1, 2] := 0;
	#rotMatrix[1, 3] := 0;
	
	// Second row
	#rotMatrix[2, 1] := 0;
	#rotMatrix[2, 2] := COS_LREAL(IN := #tempAngleRadians);
	#rotMatrix[2, 3] := - SIN_LREAL(IN := #tempAngleRadians);
	
	// Third row
	#rotMatrix[3, 1] := 0;
	#rotMatrix[3, 2] := SIN_LREAL(IN := #tempAngleRadians);
	#rotMatrix[3, 3] := COS_LREAL(IN := #tempAngleRadians);
END_FUNCTION

FUNCTION_BLOCK "LKinCtrl_MC_MovePath"
TITLE = LKinCtrl_MC_MovePath
{ S7_Optimized_Access := 'TRUE' }
AUTHOR : 'handling.team.automation@siemens.com'
FAMILY : LKinCtrl
VERSION : 5.0
//Core function block of LKinCtrl library:
//executes path motion provided by PathData command list
   VAR_INPUT 
      execute : Bool;   // rising edge starts action once
      stop : Bool;   // abort path motion
      interrupt : Bool;   // interrupt path motion
      reset : Bool;   // reset FB / acknowledge errors
      sequenceMode : Int;   // activate sequence mode (0) / single step mode (1)
      pathTransition : DInt;   // initial transition configuration for new path motion (1: use bufferMode and transitionParameter)
      bufferMode : DInt := 1;   // inital bufferMode for new path motion
      transitionParameter : Array[1..5] of LReal := [-1.0];   // initial transitionParameter for new path motion
      configuration : "LKinCtrl_typeConfiguration";   // configuration structure
      abortMeasurementCmd : Bool;   // TRUE: abort active command if measurement command
   END_VAR

   VAR_OUTPUT 
      done { ExternalWritable := 'False'} : Bool;   // TRUE: Commanded functionality has been completed successfully
      busy { ExternalWritable := 'False'} : Bool;   // TRUE: FB is not finished and new output values can be expected
      active { ExternalWritable := 'False'} : Bool;   // FB in control of axesGroup / kinematic in motion
      commandAborted { ExternalWritable := 'False'} : Bool;   // TRUE: Commanded functionality has been aborted by another command
      error { ExternalWritable := 'False'} : Bool;   // TRUE: An error occurred during the execution of the FB
      status { ExternalWritable := 'False'} : Word := #STATUS_NO_CALL;   // status of the FB
      diagnostics { ExternalWritable := 'False'} : "LKinCtrl_typeMovePathDiagnostics";   // diagnostics information of FB
      activePathData { ExternalWritable := 'False'} : String["LKINCTRL_LENGTH_OF_PATHDATA_NAME"];   // name of actual PathData
      activeCmdNo { ExternalWritable := 'False'} : DInt := 0;   // number of actual PathData set
      remainingDistanceActCmd { ExternalWritable := 'False'} : LReal;   // remaining distance of actual PathData set
      readyForNextPath { ExternalWritable := 'False'} : Bool := TRUE;   // TRUE: Next PathData can be triggered
      activeUserFrames { ExternalWritable := 'False'; S7_HiddenAssignment := 'Show'} : Array["LKINCTRL_CS_NO_OF_FIRST_USER_FRAME".."LKINCTRL_CS_NO_OF_LAST_USER_FRAME"] of "LKinCtrl_typeFrame";   // Currently acitve user frames
   END_VAR

   VAR_IN_OUT 
      axesGroup {InstructionName := 'TO_Kinematics'; LibVersion := '9.0'} : TO_Kinematics;   // reference to the axesGroup
      pathData : "LKinCtrl_typePathData";   // reference to the PathData
      pointTable : Array[*] of "LKinCtrl_typePoint";   // reference to point table
      flags : Array[*] of Bool;   // boolean defined by setFlags in PathCommand
      valueFlags : Array[*] of LReal;   // value defined by valueFlags in PathCommand
   END_VAR

   VAR 
      statExecuteOld { ExternalAccessible := 'False'; ExternalVisible := 'False'; ExternalWritable := 'False'} : Bool;   // old value of 'execute' input for edge detection
      statStopOld { ExternalAccessible := 'False'; ExternalVisible := 'False'; ExternalWritable := 'False'} : Bool;   // old value of 'stop' input for edge detection
      statInterruptOld { ExternalAccessible := 'False'; ExternalVisible := 'False'; ExternalWritable := 'False'} : Bool;   // old value of 'interrupt' input for edge detection
      statResetOld { ExternalAccessible := 'False'; ExternalVisible := 'False'; ExternalWritable := 'False'} : Bool;   // old value of 'reset' input for edge detection
      statDone { ExternalAccessible := 'False'; ExternalVisible := 'False'; ExternalWritable := 'False'} : Bool;   // static value for output 'done'
      statBusy { ExternalAccessible := 'False'; ExternalVisible := 'False'; ExternalWritable := 'False'} : Bool;   // static value for output 'busy'
      statCommandAborted { ExternalAccessible := 'False'; ExternalVisible := 'False'; ExternalWritable := 'False'} : Bool;   // static value for output 'commandAborted'
      statError { ExternalAccessible := 'False'; ExternalVisible := 'False'; ExternalWritable := 'False'} : Bool;   // static value for output 'error'
      statStatus { ExternalAccessible := 'False'; ExternalVisible := 'False'; ExternalWritable := 'False'} : Word := #STATUS_NO_CALL;   // static value for output 'status'
      statErrorID { ExternalAccessible := 'False'; ExternalVisible := 'False'; ExternalWritable := 'False'} : Word;   // static value for diagnostics output: errorID
      statSubfunctionStatus { ExternalAccessible := 'False'; ExternalVisible := 'False'; ExternalWritable := 'False'} : Word;   // status or return value of called FBs, FCs and system blocks
      statReadyForNextPath { ExternalAccessible := 'False'; ExternalVisible := 'False'; ExternalWritable := 'False'} : Bool := TRUE;   // static value for output 'readyForNextPath'
      statActivePathData { ExternalAccessible := 'False'; ExternalVisible := 'False'; ExternalWritable := 'False'} : String["LKINCTRL_LENGTH_OF_PATHDATA_NAME"];   // static value for active path data name
      statActiveCmdNo { ExternalAccessible := 'False'; ExternalVisible := 'False'; ExternalWritable := 'False'} : DInt;   // static value for output "activeCmdNo"
      statRemainingDistanceActCmd { ExternalAccessible := 'False'; ExternalVisible := 'False'; ExternalWritable := 'False'} : LReal;   // static value for output "remainingDistActCmd"
      statInterruptedAtStart { ExternalAccessible := 'False'; ExternalVisible := 'False'; ExternalWritable := 'False'} : Bool;   // static to store if interrupt was executed at start of path
      statStateExecution { ExternalAccessible := 'False'; ExternalVisible := 'False'; ExternalWritable := 'False'} : DInt := #EX_NO_PROCESSING;   // state in the state machine of the FB
      statStatePreBuffering { ExternalAccessible := 'False'; ExternalVisible := 'False'; ExternalWritable := 'False'} : DInt := #PB_NO_PROCESSING;   // state in the state machine of the FB
      statDebugState { ExternalAccessible := 'False'; ExternalVisible := 'False'; ExternalWritable := 'False'} : Bool;   // static variable to debug IF state machine if needed
      statEmptyDiagnostics { ExternalAccessible := 'False'; ExternalVisible := 'False'; ExternalWritable := 'False'; S7_SetPoint := 'False'} : "LKinCtrl_typeMovePathDiagnostics";   // empty diagnostics information (for initialization purposes only)
      statPreBufferCmdCtr { ExternalAccessible := 'False'; ExternalVisible := 'False'; ExternalWritable := 'False'} : Int;   // static counter to run FB LKinCtrl_PreBuffer multiple times
      statLastCmdIdPathdata { ExternalAccessible := 'False'; ExternalVisible := 'False'; ExternalWritable := 'False'} : DInt;   // static value to store last detected cmd in PathData
      statStoreInterruptStateExecution { ExternalAccessible := 'False'; ExternalVisible := 'False'; ExternalWritable := 'False'} : DInt;   // static store variable for state machine status on interrupt
      statPathDataIdentifier { ExternalAccessible := 'False'; ExternalVisible := 'False'; ExternalWritable := 'False'} : USInt;   // static to identify PathDatas independent of given name
      statWrittenActiveCmdNo { ExternalAccessible := 'False'; ExternalVisible := 'False'; ExternalWritable := 'False'} : DInt;   // static to store the last written active command number
      statMCExecuteWasDone { ExternalAccessible := 'False'; ExternalVisible := 'False'; ExternalWritable := 'False'} : Bool;   // static to store done output of MC_Execute in case of wait flags at end of path
      statExecutionWaitSingleStep { ExternalAccessible := 'False'; ExternalVisible := 'False'; ExternalWritable := 'False'} : Bool;   // static bit to wait for execution due to sequenceMode
      statPauseExecution { ExternalAccessible := 'False'; ExternalVisible := 'False'; ExternalWritable := 'False'} : Bool;   // static bit to wait for execution due to wait time or tool ommands running
      statWaitMain { ExternalAccessible := 'False'; ExternalVisible := 'False'; ExternalWritable := 'False'} : Bool;   // static bit to wait for execution due to wait flags
      statWaitValueMain { ExternalAccessible := 'False'; ExternalVisible := 'False'; ExternalWritable := 'False'} : Bool;   // static bit to wait for execution due to wait value flags
      statPreBufferError { ExternalAccessible := 'False'; ExternalVisible := 'False'; ExternalWritable := 'False'} : Bool;   // static to store error output of prebuffer
      statPreBufferedPathDataNameOld { ExternalAccessible := 'False'; ExternalVisible := 'False'; ExternalWritable := 'False'} : String["LKINCTRL_LENGTH_OF_PATHDATA_NAME"];   // static to store old PathDataName in PathDataPreBuffered
      statPreBufferedCmdIdOld { ExternalAccessible := 'False'; ExternalVisible := 'False'; ExternalWritable := 'False'} : DInt;   // static to store old cmdId value from PathDataPreBuffered
      statPathDataPreBufferAddPointerOld { ExternalAccessible := 'False'; ExternalVisible := 'False'; ExternalWritable := 'False'} : Int;   // old value of 'addPointer' in PathDataPreBuffer
      statSetFlagsBufferWriteBufferElement_old { ExternalAccessible := 'False'; ExternalVisible := 'False'; ExternalWritable := 'False'} : Int;   // static to store old setFlagsBuffer write element pointer value
      statFirstCycle { ExternalAccessible := 'False'; ExternalVisible := 'False'; ExternalWritable := 'False'} : Bool;   // static indicating first cycle
      statInitStartPos { ExternalAccessible := 'False'; ExternalVisible := 'False'; ExternalWritable := 'False'} : Bool;   // static start position
      statIsMeasurementCmd { ExternalAccessible := 'False'; ExternalVisible := 'False'; ExternalWritable := 'False'} : USInt;   // output value of ExecuteKinMotionCmd
      statStateOld { ExternalAccessible := 'False'; ExternalVisible := 'False'; ExternalWritable := 'False'} : DInt;   // static to store the last execution state
      statAbortOld { ExternalAccessible := 'False'; ExternalVisible := 'False'; ExternalWritable := 'False'} : Bool := false;   // static bit to store aborted state
      statActiveCmdNoOld { ExternalAccessible := 'False'; ExternalVisible := 'False'; ExternalWritable := 'False'} : DInt;   // old value of activeCmdNo
      statFlagsBuffer { ExternalAccessible := 'False'; ExternalVisible := 'False'; ExternalWritable := 'False'} : Struct   // buffer to store flag information for past and actual commands
         writeBufferElement { ExternalAccessible := 'False'; ExternalVisible := 'False'; ExternalWritable := 'False'} : Int := 1;   // pointer on entry to be written
         bufferElement { ExternalAccessible := 'False'; ExternalVisible := 'False'; ExternalWritable := 'False'; S7_SetPoint := 'False'} : Array[1.."LKINCTRL_NO_OF_SETFLAGS_BUFFER_ELEMENTS"] of "LKinCtrl_typeFlagBufferElement";   // flag information for one specific command (see cmdId)
      END_STRUCT;
      statPathDataPreBuffered { ExternalAccessible := 'False'; ExternalVisible := 'False'; ExternalWritable := 'False'; S7_SetPoint := 'False'} : "LKinCtrl_typePathData_PreBuf" := ((), [((), (), (), (), (), (), (), ([()], [()], [()], ()), (((), (), (), ()), ((), (), (), ()), (), (), [-1.0], (), (), ((), (), [()]), ((), ()), (()), ((), (), [()], (), (), (), ()), ((), (), ()), (([()], (), (), ()), ([()], (), (), ()))), [((), (), ()), ((), (), ()), ((), (), ())], [((), (), (), ()), ((), (), (), ()), ((), (), (), ()), ((), (), (), ())], [6(TRUE)]), ((), (), (), (), (), (), (), ([()], [()], [()], ()), (((), (), (), ()), ((), (), (), ()), (), (), [-1.0], (), (), ((), (), [()]), ((), ()), (()), ((), (), [()], (), (), (), ()), ((), (), ()), (([()], (), (), ()), ([()], (), (), ()))), [((), (), ()), ((), (), ()), ((), (), ())], [((), (), (), ()), ((), (), (), ()), ((), (), (), ()), ((), (), (), ())], [6(TRUE)]), ((), (), (), (), (), (), (), ([()], [()], [()], ()), (((), (), (), ()), ((), (), (), ()), (), (), [-1.0], (), (), ((), (), [()]), ((), ()), (()), ((), (), [()], (), (), (), ()), ((), (), ()), (([()], (), (), ()), ([()], (), (), ()))), [((), (), ()), ((), (), ()), ((), (), ())], [((), (), (), ()), ((), (), (), ()), ((), (), (), ()), ((), (), (), ())], [6(TRUE)]), ((), (), (), (), (), (), (), ([()], [()], [()], ()), (((), (), (), ()), ((), (), (), ()), (), (), [-1.0], (), (), ((), (), [()]), ((), ()), (()), ((), (), [()], (), (), (), ()), ((), (), ()), (([()], (), (), ()), ([()], (), (), ()))), [((), (), ()), ((), (), ()), ((), (), ())], [((), (), (), ()), ((), (), (), ()), ((), (), (), ()), ((), (), (), ())], [6(TRUE)]), ((), (), (), (), (), (), (), ([()], [()], [()], ()), (((), (), (), ()), ((), (), (), ()), (), (), [-1.0], (), (), ((), (), [()]), ((), ()), (()), ((), (), [()], (), (), (), ()), ((), (), ()), (([()], (), (), ()), ([()], (), (), ()))), [((), (), ()), ((), (), ()), ((), (), ())], [((), (), (), ()), ((), (), (), ()), ((), (), (), ()), ((), (), (), ())], [6(TRUE)])], (), (), ());   // preBuffered PathData elements (internal buffer of path motion commands)
      statPathDataElementPreBuffered { ExternalAccessible := 'False'; ExternalVisible := 'False'; ExternalWritable := 'False'; S7_SetPoint := 'False'} : "LKinCtrl_typePathDataElement_PreBuf" := ((), (), (), (), (), (), (), ([()], [()], [()], ()), (((), (), (), ()), ((), (), (), ()), (), (), [-1.0], (), (), ((), (), [()]), ((), ()), (()), ((), (), [()], (), (), (), ()), ((), (), ()), (([()], (), (), ()), ([()], (), (), ()))), [((), (), ()), ((), (), ()), ((), (), ())], [((), (), (), ()), ((), (), (), ()), ((), (), (), ()), ((), (), (), ())], [6(TRUE)]);   // PathData element  to be executed by FB_ExecutePathMotion
      statWaitFlags { ExternalAccessible := 'False'; ExternalVisible := 'False'; ExternalWritable := 'False'} : Struct   // static struct to store wait flag information
         waitCtr { ExternalAccessible := 'False'; ExternalVisible := 'False'; ExternalWritable := 'False'} : Int;   // counter for number of wait flags in one command
         waitFlag { ExternalAccessible := 'False'; ExternalVisible := 'False'; ExternalWritable := 'False'} : Array[1.."LKINCTRL_NO_OF_CMD_SETFLAGS"] of Int;   // flag number as identifier for flag active as wait flag
      END_STRUCT;
      statWaitValueFlags { ExternalAccessible := 'False'; ExternalVisible := 'False'; ExternalWritable := 'False'} : Struct   // static struct to store wait valueFlag information
         waitCtr { ExternalAccessible := 'False'; ExternalVisible := 'False'; ExternalWritable := 'False'} : Int;   // counter for number of wait flags in one command
         waitFlag { ExternalAccessible := 'False'; ExternalVisible := 'False'; ExternalWritable := 'False'} : Array[1.."LKINCTRL_NO_OF_CMD_VALUEFLAGS"] of Int;   // flag number as identifier for flag active as wait valueFlag
      END_STRUCT;
      statEmptyPathDataElementPreBuffered { ExternalAccessible := 'False'; ExternalVisible := 'False'; ExternalWritable := 'False'; S7_SetPoint := 'False'} : "LKinCtrl_typePathDataElement_PreBuf" := ((), (), (), (), (), (), (), ([()], [()], [()], ()), (((), (), (), ()), ((), (), (), ()), (), (), [-1.0], (), (), ((), (), [()]), ((), ()), (()), ((), (), [()], (), (), (), ()), ((), (), ()), (([()], (), (), ()), ([()], (), (), ()))), [((), (), ()), ((), (), ()), ((), (), ())], [((), (), (), ()), ((), (), (), ()), ((), (), (), ()), ((), (), (), ())], [6(TRUE)]);   // static for empty pre buffer element
      statEmptyFlagBufferElement { ExternalAccessible := 'False'; ExternalVisible := 'False'; ExternalWritable := 'False'; S7_SetPoint := 'False'} : "LKinCtrl_typeFlagBufferElement";   // static for empty flagBuffer element
      instLKinCtrl_SetFlagCtrl { ExternalAccessible := 'False'; ExternalVisible := 'False'; ExternalWritable := 'False'; S7_SetPoint := 'False'} : "LKinCtrl_SetFlagCtrl";   // instance of flag controls for setFlags
      instLKinCtrl_ValueFlagCtrl { ExternalAccessible := 'False'; ExternalVisible := 'False'; ExternalWritable := 'False'; S7_SetPoint := 'False'} : "LKinCtrl_ValueFlagCtrl";   // instance of flag controls for valueFlags
      instLKinCtrl_PreBuffer { ExternalAccessible := 'False'; ExternalVisible := 'False'; ExternalWritable := 'False'; S7_SetPoint := 'False'} : "LKinCtrl_PreBuffer";
      instLKinCtrl_MC_ExecuteKinMotionCmd { ExternalAccessible := 'False'; ExternalVisible := 'False'; ExternalWritable := 'False'; S7_SetPoint := 'False'} : "LKinCtrl_MC_ExecuteKinMotionCmd";
   END_VAR

   VAR_TEMP 
      tempExecute : Bool;   // Temporary value for input 'execute'
      tempStop : Bool;   // Temporary value for input 'stop'
      tempInterrupt : Bool;   // Temporary value for input 'interrupt'
      tempReset : Bool;   // Temporary value for input 'stop'
      tempSequenceMode : Int;   // Temporary value for input 'sequenceMode'
      tempCtr : DInt;   // Temporary command counter
      tempPreBufferPtrOk : Bool;   // Temporary bit for pointer checks
      tempExecutionWaiting : Bool;   // Temporary bit to disable triggering commands
      tempKinematicsStatusWord : DWord;   // Temporary copy of TO Kinematics status word
      tempMotionQueueCommands : DInt;   // Temporary copy of TO Kinematics number of commands in motion queue
      tempExecCtr : DInt;   // Temporary counter
      tempWaitFlagFound : Bool;   // Temporary bit to signal a wait flag was found
      tempFlagBufferElement : "LKinCtrl_typeFlagBufferElement";   // Temporary storing for a flagBuffer element
      tempAbortMeasurementCmd : Bool;   // Temporary value for input 'abortMeasurementCmd'
      tempStopMeasure : Bool;   // Temporary value to trigger executer stop
   END_VAR

   VAR CONSTANT 
      EX_NO_PROCESSING : Int := 0;   // state machine constant
      EX_RESETTING : Int := 5;   // state machine constant
      EX_INTERRUPT_AT_START : Int := 10;   // state machine constant
      EX_CONTINUE_AT_START : Int := 11;   // state machine constant
      EX_GET_CMD : Int := 30;   // state machine constant
      EX_TRIGGERING_CMD : Int := 50;   // state machine constant
      EX_TRIGGERED_CMD : Int := 55;   // state machine constant
      EX_INTERRUPTING : Int := 70;   // state machine constant
      EX_INTERRUPTED : Int := 75;   // state machine constant
      EX_CONTINUEING : Int := 77;   // state machine constant
      EX_CONTINUED : Int := 78;   // state machine constant
      EX_STOPPING : Int := 80;   // state machine constant
      EX_STOPPED_STATE : Int := 85;   // state machine constant
      EX_ERROR_STATE : Int := 90;   // state machine constant
      EX_ALL_TRIGGERED : Int := 100;   // state machine constant
      EX_ABORT_MEAS_CMD : Int := 105;   // state machine constant
      EX_MEAS_CMD_ABORTED : Int := 110;   // state machine constant
      PB_NO_PROCESSING : Int := 0;   // state machine constant
      PB_ENABLED : Int := 10;   // state machine constant
      PB_OFF_COMP : Int := 15;   // state machine constant
      PB_DISABLED : Int := 20;   // state machine constant
      STATUS_EXECUTION_FINISHED : Word := 16#0000;   // status execution finished without errors
      STATUS_NO_CALL : Word := 16#7000;   // status no job being currently processed
      STATUS_FIRST_CALL : Word := 16#7001;   // status first call after incoming new job (rising edge 'execute')
      STATUS_SUBSEQUENT_CALL : Word := 16#7002;   // status subsequent call during active processing without further details
      STATUS_FB_RESETTING : Word := 16#7010;   // status FB resetting
      STATUS_WAITING_FOR_PREBUFFERED_CMD : Word := 16#7070;   // status waiting for new command in PathData_Prebuffered
      STATUS_PREBUFFERED_FULL : Word := 16#7071;   // status internal cmd buffer filled completely
      STATUS_CMD_LIN_ACTIVE : Word := 16#7301;   // status linear motion command active at axesgroup
      STATUS_CMD_CIRC_ACTIVE : Word := 16#7302;   // status circular motion command active at axesgroup
      STATUS_PATHMOTION_INTERRUPTED : Word := 16#7303;   // status path motion interrupted
      STATUS_PATHMOTION_STOPPING : Word := 16#7304;   // status path motion stopping
      STATUS_READYFORNEXTPATH : Word := 16#7305;   // status FB ready for next path execution
      STATUS_PATHMOTION_RUNNING : Word := 16#7306;   // status path motion running
      STATUS_EXECUTION_WAITING : Word := 16#7307;   // status path execution waiting due to wait flag, wait time or single step mode
      STATUS_CMD_MOVE_DIRECT_ACTIVE : Word := 16#7308;   // status move direct motion command active at axesgroup
      STATUS_STOP_DUE_TO_ERROR : Word := 16#7309;   // status kinematics is stopped due to an error in FB Executer
      STATUS_CMD_CONFIGURATION_ACTIVE : Word := 16#730A;   // status configuration command active at axesgroup
      STATUS_COMMAND_ABORTED : Word := 16#7FFF;   // status commanded functionality has been aborted by another command
      ERR_UNDEFINED_STATE : Word := 16#8600;   // error due to an undefined state in state machine
      ERR_EXECUTE_KINMOTIONCMD : Word := 16#8201;   // error due to error in FB LKinCtrl_ExecuteKinMotionCmd
      ERR_WRONG_SEQUENCEMODE : Word := 16#8203;   // error due to invalid sequenceMode on input
      ERR_PATHDATA_PARAMETERS : Word := 16#8204;   // error due to malconfiguration in motion command parameters
      ERR_OFFSET_CALCULATION : Word := 16#8205;   // error due to calculation error in offset compensation
      ERR_ERROR_STILL_PENDING : Word := 16#8207;   // error due to previous not acknowledged error (reset MovePath to acknowledge)
      ERR_SET_FLAG_CONTROL : Word := 16#8208;   // error due to error in set flag control FB
      ERR_VALUE_FLAG_CONTROL : Word := 16#8209;   // error due to error in value flag control FB
      ERR_TRIGGER_NOT_POSSIBLE : Word := 16#820A;   // error due to new execute not possible
      INTERRUPT_AT_START : Bool := FALSE;   // interrupt at start of new path to preload commands
      NO_OF_COMMANDS_PRELOADING : USInt := 3;   // number of commands to be preloaded
      CONTINUE_AT_START : Bool := TRUE;   // continue at start of new path
   END_VAR


BEGIN
	//==========================================================================================
	// SIEMENS AG
	// (c)Copyright 2020 All Rights Reserved
	//------------------------------------------------------------------------------------------
	// Library: LKinCtrl
	// Tested with: S7-1517T-3 PN/DP
	// Engineering: TIA Portal V16
	// Restrictions: ---
	// Requirements: S7-1500T FW 2.8
	// Functionality: LKinCtrl_MC_MovePath
	// The FB is executing a sequence to drive a path defined by the user in form of a
	// command list of points and motion commands.
	//
	// Support: tech.team.motioncontrol@siemens.com
	// Note: Parameter comments are only available in language 'English (United States)'
	//------------------------------------------------------------------------------------------
	// Change log table:
	// Version    Date          Expert in charge    Changes applied
	// 01.00.00   06.02.2018    JR                  First release version v1.0
	// 02.00.00   18.04.2019    JR / FR             V2.0
	// 02.01.00   28.05.2019    JR / FR             V2.1 for LKinLang
	// 02.02.00   28.01.2020    JR / FR             V2.2: Added valueFlags and flagOnlyCmd 
	// 02.02.01   07.02.2020    FR / DF             V2.2.1: Disable Prebuffer when MovePath is stopping/reseting/(done)
	// 02.02.02   12.02.2020    FR                  Fix for loops using wrong flag constant
	// 02.03.00   18.03.2020    FR                  Rework Flag FBs; Fix for interrupt/continue
	// 02.04.00   25.03.2020    FR                  Added preprocessing stop for LKinLang
	// 02.04.01   07.05.2020    FR                  Fix 360° circle with circMode 3
	// 02.04.02   16.07.2020    FR                  Several bugfixes
	// 03.00.00   04.08.2020    FR                  Added MoveDirect and ConveyorTracking; V16/FW2.8.2 required!
	// 03.00.01   06.08.2020    FR                  Bugfix
	// 03.00.02   19.10.2020    FR                  Updated ContourOffset; Updated FlagControl; Bugfixes
	// 03.00.03   23.11.2020    FR                  Updated ContourOffset; Fix in MC_ExecuteKinMotionCmd
	// 03.00.05   01.06.2021    FR                  Fixes in FlagCtrl FBs
	// 03.01.00   01.07.2021    FR                  Added Frame, Tool and Zone commands; code cleanup
	// 03.01.02   20.10.2021    FR                  Changed interrupt/Continue handling & Bugfixes
	// 03.01.03   16.11.2021    FR                  Updated contourOffset; Bugfixes
	// 03.02.00   16.02.2022    FR                  Bugfix for Interrupt & Continue, Bugfix for Flags, Option to execute multiple commands per cycle
	// 03.03.00   17.08.2022    FR                  Added orientation dynamics to pathData, New FlagModes, Bugfixes
	// 04.00.00   26.01.2023    FR                  Support MC Version 7.0, Added PointTable
	// 04.00.01   23.02.2023    FR                  Updated valid bits, Bugfixes
	// 04.01.00   02.02.2024    FR / AH             Structural changes
	// 04.01.01   07.02.2024    AH                  Bugfix
	// 04.01.02   09.02.2024    FR                  Bugfixes in command preparation
	// 04.01.03   11.04.2024    FR                  Bugfixes
	// 04.01.05   02.05.2024    FR                  Bugfixes
	// 04.02.00   11.07.2024    AH                  Added measurement functionality - additional input "abortMeasurementCmd" & Bugfixes
	// 05.00.00   05.09.2024    FR                  Switch pathData from variant to "LKinCtrl_typePathData"
	//===========================================================================================
	
	// Work with temporary value / create process image
	#tempExecute := #execute;
	#tempStop := #stop;
	#tempInterrupt := #interrupt;
	#tempReset := #reset;
	#tempSequenceMode := #sequenceMode;
	#tempKinematicsStatusWord := #axesGroup.StatusWord;
	#tempMotionQueueCommands := #axesGroup.StatusMotionQueue.NumberOfCommands;
	#tempAbortMeasurementCmd := #abortMeasurementCmd;
	
	// Reset first cycle
	#statFirstCycle := FALSE;
	
	
	REGION TRIGGERING
	  //-----------------------------------------------------------------------------
	  // check for SEQUENCEMODE to be activated
	  //-----------------------------------------------------------------------------
	  IF #tempSequenceMode = 1 THEN
	    // set execution wait bit to stop cmds from being executed (wait in EX_TRIGGERING_CMD)
	    #statExecutionWaitSingleStep := TRUE;
	    // check for incorrect sequenceMode to be selected
	  ELSIF (#tempSequenceMode <> 0 AND #tempSequenceMode <> 1)
	    // only check if execution is triggered
	    AND #tempExecute = TRUE
	  THEN
	    // set status accordingly
	    #statStatus := #ERR_WRONG_SEQUENCEMODE;
	    // set execution state machine
	    #statStateExecution := #EX_ERROR_STATE;
	  END_IF;
	  //===========================================================================================
	  
	  //-----------------------------------------------------------------------------
	  // check for rising edge of STOP input
	  //-----------------------------------------------------------------------------
	  IF (#tempStop = TRUE) AND (#statStopOld = FALSE) THEN
	    // perform stop procedure
	    #statStateExecution := #EX_STOPPING;
	    // FR 08.04.2020: Set status and bits here to avoid return when status = STATUS_NO_CALL
	    #statStatus := #STATUS_PATHMOTION_STOPPING;
	    #statDone := FALSE;
	    #statBusy := TRUE;
	    #statCommandAborted := FALSE;
	    #statError := FALSE;
	    #statErrorID := 16#0;
	    //===========================================================================================
	    
	    //-----------------------------------------------------------------------------
	    // check for rising edge of INTERRUPT input
	    //-----------------------------------------------------------------------------
	    // FR 17.03.2020: Added "statDone" to condition
	    // FR 09.04.2020: Added stopping status to condition
	  ELSIF (#tempInterrupt = TRUE) AND (#statInterruptOld = FALSE)
	    AND (#statDone = FALSE)
	    AND (#statError = FALSE)
	    AND #statStatus <> #STATUS_PATHMOTION_STOPPING
	    AND #statStatus <> #STATUS_COMMAND_ABORTED
	    AND #statStatus <> #STATUS_NO_CALL
	  THEN
	    
	    // FR 11.03.2020: Only save state in some cases
	    IF #statStateExecution < #EX_INTERRUPTING
	      OR #statStateExecution > #EX_CONTINUED
	    THEN
	      // store states of interruption for later continue
	      #statStoreInterruptStateExecution := #statStateExecution;
	    END_IF;
	    
	    // perform interrupt procedure
	    #statStateExecution := #EX_INTERRUPTING;
	    
	    //-----------------------------------------------------------------------------
	    // check for rising edge of RESET input
	    //-----------------------------------------------------------------------------
	  ELSIF (#tempReset = TRUE) AND (#statResetOld = FALSE)
	    AND (#statBusy = FALSE) // interlock reset during execution
	  THEN
	    // perform reset procedure
	    #statStateExecution := #EX_RESETTING;
	    #statStatePreBuffering := #PB_NO_PROCESSING;
	    // set status accordingly
	    #statStatus := #STATUS_FB_RESETTING;
	    
	    
	    //-----------------------------------------------------------------------------
	    // check for rising edge of EXECUTE input
	    //-----------------------------------------------------------------------------
	  ELSIF (#tempExecute = TRUE) AND (#statExecuteOld = FALSE)
	    AND (#tempStop = FALSE) AND (#tempInterrupt = FALSE)
	  THEN
	    //-----------------------------------------------------------------------------
	    // ERROR on start
	    //-----------------------------------------------------------------------------
	    // check for state machine to be in error state from previous (not acknowledged) error
	    IF #statStateExecution = #EX_ERROR_STATE THEN
	      // State machine - do not start cmd execution and wait in error state
	      #statStateExecution := #EX_ERROR_STATE;
	      #statStatePreBuffering := #PB_NO_PROCESSING;
	      
	      // check for error already detected before execute in this cycle (e.g. wrong sequenceMode / other faulty inputs)
	      IF #statStatus = #ERR_WRONG_SEQUENCEMODE THEN
	        #statBusy := FALSE; // reset statBusy to avoid interlock of reset
	      ELSE
	        #statStatus := #ERR_ERROR_STILL_PENDING; // set status to set error bit
	      END_IF;
	      //===========================================================================================
	      
